       // xtal handling lift swivel in      
         "CM_ITL_IO"(ADR := 68,
             KYD_ON := "KYD".XT_HDL_SW_IN AND "PDI".MP_ENB_K9,
             KYD_OFF := NOT "KYD".XT_HDL_SW_IN OR NOT "PDI".MP_ENB_K9,
             AUTO := "DV".XT_HDL_SEQ_MOD,
             DC_ON:= "DC".XT_HDL_SW_IN AND "PDI".MP_ENB_K9,
             CON1 := "PDI".EMO AND "PDI".EMS,
             CON2 := NOT "FLT".XT_HDL_SW_ERR,
             CON3 := "PDI".LS_XT_HDL_SW_UNLOCK AND NOT "PDI".LS_XT_HDL_SW_LOCK,
             CON4 := #REL_XT_HDL_SW_IN_OK OR "DV".MP_SERVICE,   
             CON5 := NOT "DV".LS_XT_HDL_SW_IN_POS OR "DV".MP_SERVICE,  
             CON6 := ("DIS".ACT_POS_XT_HDL_LFT>=1200.0)OR "DV".MP_SERVICE,
             CON7 := "SysLog1",                     
             CON8 := "SysLog1",   
             ITL_OUT:= "STA_ITL_CAUSE",
             LT_OUT := "LT".XT_HDL_SW_IN);  

         "LT".LS_XT_HDL_SW_IN  :=  "DV".LS_XT_HDL_SW_IN_XT_POS;
         "LT".XT_HDL_SW_IN_REL :=        "PDI".EMO AND "PDI".EMS
                              AND NOT "FLT".XT_HDL_SW_ERR
                              AND "PDI".LS_XT_HDL_SW_UNLOCK AND NOT "PDI".LS_XT_HDL_SW_LOCK
                              AND (#REL_XT_HDL_SW_IN_OK OR "DV".MP_SERVICE)   
                              AND (NOT "DV".LS_XT_HDL_SW_IN_CRU_POS OR "DV".MP_SERVICE)
                              AND (("DIS".ACT_POS_XT_HDL_LFT>=1200.0)OR "DV".MP_SERVICE);

         #REL_XT_HDL_SW_IN_OK :=  (("DIS".ACT_POS_XT_HDL_LFT>1160.0) AND ("DIS".ACT_POS_XT_HDL_SW<"CNF".XT_HDL_SW_IN_TRP_POS )) 
                               OR ("PDI".LS_XT_CLP_CON AND "PDI".LS_GCH_DOOR_OP AND NOT "PDI".LS_XT_SLID_BW) 
                               OR ("PDI".LS_HOI_TOOL_INST AND "AV".TEC_FLG_ENC_POS > 100.0)
                               OR "DV".MP_SERVICE;   

         IF "LT".XT_HDL_SW_IN THEN 
           #set_speed  := "CNF_XT_HDL_SW_LZ950".SEL_SPEED;  // swivel in 
         END_IF;
         IF "LT".XT_HDL_SW_OUT THEN 
           #set_speed  := -"CNF_XT_HDL_SW_LZ950".SEL_SPEED;  // swivel out 
         END_IF;       
         IF NOT "LT".XT_HDL_SW_IN AND NOT "LT".XT_HDL_SW_OUT THEN 
           #set_speed  := 0.0; 
         END_IF;

        // Release reference set
         "LT".XT_HDL_SW_REF_RUN  := "DV".XT_HDL_SW_SET_REF_POS; ///XT_HDL_SW.READY AND NOT XT_HDL_SW.Ref_Done; //DV.XT_HDL_SW_SET_REF_POS;
         "LT".XT_HDL_SW_REF_DONE := #XT_HDL_SW.Ref_Done OR "SY".SIM_ON;                     


         #XT_HDL_SW (Enable         := ("LT".XT_HDL_SW_IN OR "LT".XT_HDL_SW_OUT OR "LT".XT_HDL_SW_REF_RUN), 
                   Pro_start     := ("LT".XT_HDL_SW_OUT OR "LT".XT_HDL_SW_IN),   
                   Speed_ext_ovr := TRUE,   
                   Ref_Start     := "LT".XT_HDL_SW_REF_RUN,
                   Ref_reset     := FALSE,
                   Reset_error   := "KYD".XT_HDL_SW_TRIP_RES,
                   Stop          := NOT "LT".XT_HDL_SW_OUT AND NOT "LT".XT_HDL_SW_IN,
                   Profil        := "CNF_XT_HDL_SW_LZ950".Profil,
                   PM_ADR_E      := INT_TO_WORD("CNF_XT_HDL_SW_LZ950".PE_ADR),                                   
                   PM_ADR_A      := INT_TO_WORD("CNF_XT_HDL_SW_LZ950".PA_ADR),                
                   Units_per_rev := "CNF_XT_HDL_SW_LZ950".UNITS_PER_REV,                       
                   Gear_ratio    := "CNF_XT_HDL_SW_LZ950".FEED_CONST,
                   Set_vel       := #set_speed); 


        //actual motor values
        //---------------------
         "AV".XT_HDL_SW_ACT_POS   := #XT_HDL_SW.Act_pos;
         "DIS".ACT_POS_XT_HDL_SW  := "AV".XT_HDL_SW_ENC_POS;   

        //actual fault
        //---------------------
         "DIS".XT_HDL_SW_ERR_CODE := #XT_HDL_SW.Error_code;        // Fehlernummer Umrichter
         "FLT".XT_HDL_SW_ERR      := #XT_HDL_SW.Error;             // Fehlerbit Umrichter
         "FLT".XT_HDL_SW_POS_REF  := NOT "LT".XT_HDL_SW_REF_DONE;   // Antrieb nicht referenziert
         "FLT".XT_HDL_SW_SLS      := #XT_HDL_SW.LS_neg OR #XT_HDL_SW.LS_pos;  // Fehler Sicherheitsendschalter



        // xtal handling lift swivel lock    
         "PDO".XT_HDL_SW_LOCK   :=  "DV".LS_XT_HDL_SW_IN_XT_POS AND NOT "LT".XT_HDL_SW_IN AND NOT "LT".XT_HDL_SW_IN AND 
                              "PDI".LS_XT_HDL_SW_UNLOCK AND NOT "KYD".XT_HDL_SW_OUT;

        // xtal handling lift swivel unlock     
         "PDO".XT_HDL_SW_UNLOCK :=  (NOT "DV".LS_XT_HDL_SW_IN_XT_POS OR "KYD".XT_HDL_SW_OUT) AND NOT "PDI".LS_XT_HDL_SW_UNLOCK;

         #REL_XT_HDL_SW_DRV    :=  "LT".XT_HDL_SW_UNLOCKED OR
                              "SysOndelay"( DIN := ("KYD".XT_HDL_SW_OUT AND "PDI".MP_ENB_K9),
                                          SetTime := 3,                         // setp. time
                                          ActTime := #sw_lock_dly,               // act. time
                                          Tick    := "SysTick1s");                // timebase (1s)

        // light signal crystal handling swivel unlock/locked     
         "LT".XT_HDL_SW_UNLOCKED := "PDI".LS_XT_HDL_SW_UNLOCK;
         "LT".XT_HDL_SW_LOCKED   := "PDI".LS_XT_HDL_SW_LOCK;

        //----------------------------------------------------------------------
        // xtal handling slidering drive   
        //----------------------------------------------------------------------
        // xtal handling sliding drive forwards
         "CM_ITL_IO"(ADR := 71,
            KYD_ON := "KYD".XT_HDL_SLID_FW AND "PDI".MP_ENB_K9,
            KYD_OFF := NOT "KYD".XT_HDL_SLID_FW OR NOT "PDI".MP_ENB_K9,
            AUTO := "DV".XT_HDL_SEQ_MOD,
            DC_ON:= "DC".XT_HDL_SLID_FW AND "PDI".MP_ENB_K9,
            CON1 := "PDI".EMO AND "PDI".EMS,
            CON2 := "PDI".LS_XT_SLID_FW,
            CON3 := NOT "PDO".XT_HDL_SLID_BW, 
            CON4 := (("PDI".LS_UP_XT_CLP_OP OR "PDI".LS_UP_XT_CLP_PLATE) AND ("PDI".LS_LO_XT_CLP_OP OR "PDI".LS_LO_XT_CLP_PLATE) AND "DV".LS_XT_HDL_SW_IN_XT_POS AND ("DIS".ACT_POS_XT_HDL_LFT>839.0)) OR 
                     ("DV".LS_XT_HDL_SW_IN_TRP_POS AND ("DV".LS_XT_HDL_LFT_DN_POS OR ("DIS".ACT_POS_XT_HDL_LFT>1120.0))) OR "DV".LS_XT_HDL_SW_OUT_MAX_POS OR 
                      //OR
                     (NOT "PDI".LS_XT_CLP_CON AND ("DIS".ACT_POS_XT_HDL_LFT>1120.0)) OR "DV".MP_SERVICE,   
            CON5 := "SysLog1",   
            CON6 := "SysLog1",                     
            CON7 := "SysLog1",    
            CON8 := "SysLog1",   
            ITL_OUT:= "STA_ITL_CAUSE",
            LT_OUT := "LT".XT_SLID_FW);

       // controller crystal handling slider forwards  
        "PDO".XT_HDL_SLID_FW  :=  "LT".XT_SLID_FW;             
        "LT".XT_SLID_FW_REL   :=      "PDI".EMO AND "PDI".EMS 
                              AND "PDI".LS_XT_SLID_FW 
                              AND NOT "PDO".XT_HDL_SLID_BW
                              AND ((("PDI".LS_UP_XT_CLP_OP OR "PDI".LS_UP_XT_CLP_PLATE) AND ("PDI".LS_LO_XT_CLP_OP OR "PDI".LS_LO_XT_CLP_PLATE) AND "DV".LS_XT_HDL_SW_IN_XT_POS AND ("DIS".ACT_POS_XT_HDL_LFT>839.0))
                                     OR ("DV".LS_XT_HDL_SW_IN_TRP_POS AND ("DV".LS_XT_HDL_LFT_DN_POS OR ("DIS".ACT_POS_XT_HDL_LFT>1120.0)))  OR "DV".LS_XT_HDL_SW_OUT_MAX_POS OR 
                                     // OR
                                     (NOT "PDI".LS_XT_CLP_CON AND ("DIS".ACT_POS_XT_HDL_LFT>1120.0)) OR "DV".MP_SERVICE);                           

       // xtal handling sliding drive backwards 
        "CM_ITL_IO"(ADR := 72,
             KYD_ON := "KYD".XT_HDL_SLID_BW AND "PDI".MP_ENB_K9,
            KYD_OFF := NOT "KYD".XT_HDL_SLID_BW OR NOT "PDI".MP_ENB_K9,
            AUTO := "DV".XT_HDL_SEQ_MOD,
            DC_ON:= "DC".XT_HDL_SLID_BW AND "PDI".MP_ENB_K9,
            CON1 := "PDI".EMO AND "PDI".EMS,
            CON2 := "PDI".LS_XT_SLID_BW,
            CON3 := NOT "PDO".XT_HDL_SLID_FW, 
            CON4 := #REL_XT_CLP_POS_OK,   
            CON5 := "SysLog1",   
            CON6 := "SysLog1",                     
            CON7 := "SysLog1",    
            CON8 := "SysLog1",   
            ITL_OUT:= "STA_ITL_CAUSE",
            LT_OUT := "LT".XT_SLID_BW);

       // controller crystal handling slider backwards  
        "PDO".XT_HDL_SLID_BW  := "LT".XT_SLID_BW; 
        "LT".XT_SLID_BW_REL   :=     "PDI".EMO AND "PDI".EMS 
                            AND "PDI".LS_XT_SLID_BW 
                            AND NOT "PDO".XT_HDL_SLID_FW
                            AND #REL_XT_CLP_POS_OK;  

        #REL_XT_CLP_POS_OK :=  (NOT "PDI".LS_XT_CLP_CON  AND ("DV".LS_XT_HDL_LFT_DN_POS OR ("DIS".ACT_POS_XT_HDL_LFT>620.0)))        // without clamp
                           OR ("PDI".LS_XT_CLP_CON AND (("PDI".LS_UP_XT_CLP_CL AND "PDI".LS_LO_XT_CLP_CL) OR ("PDI".LS_UP_XT_CLP_SAVE AND "PDI".LS_LO_XT_CLP_SAVE) OR "DV".LS_XT_HDL_SW_IN_TRP_POS) 
                           AND "PDI".LS_XT_SLID_BW AND "PDI".LS_XT_TILT_90 AND ("DIS".ACT_POS_XT_HDL_LFT>620.0))   // takeover cystal 
                           OR (NOT "PDI".LS_XT_TILT_75 AND "DV".LS_XT_ACP_LFT_UPR_POS) // lift up to 1550mm position ready to swivel out to 56?
                           OR "DV".LS_XT_HDL_SW_OUT_MAX_POS
                           OR "DV".MP_SERVICE;          

       //light signal for positions  
        "LT".LS_XT_SLID_FW       :=   NOT "PDI".LS_XT_SLID_FW AND NOT "PDI".LS_XT_SLID_MID  AND "PDI".LS_XT_SLID_BW;          
        "LT".LS_XT_SLID_MID      :=   "PDI".LS_XT_SLID_MID AND "PDI".LS_XT_SLID_FW AND "PDI".LS_XT_SLID_BW;           
        "LT".LS_XT_SLID_BW       :=   NOT "PDI".LS_XT_SLID_BW AND "PDI".LS_XT_SLID_FW AND NOT "PDI".LS_XT_SLID_MID;         


       //----------------------------------------------------------------------
       // xtal handling tilt drive       
       //---------------------------------------------------------------------- 
       // xtal handling tilt drive forwards (to 75?
        "CM_ITL_IO"(ADR := 73,
            KYD_ON := "KYD".XT_CLP_TILT_75 AND "PDI".MP_ENB_K9,
            KYD_OFF := NOT "KYD".XT_CLP_TILT_75 OR NOT "PDI".MP_ENB_K9,
            AUTO := "DV".XT_HDL_SEQ_MOD,
            DC_ON:= "DC".XT_CLP_TILT_75 AND "PDI".MP_ENB_K9,
            CON1 := "PDI".EMO AND "PDI".EMS,
            CON2 := NOT "PDI".LS_XT_TILT_75,
            CON3 := NOT "PDO".XT_CLP_TILT_BW, 
            CON4 := #REL_XT_CLP_TILT_POS_OK OR "DV".MP_SERVICE,                
            CON5 := "SysLog1",   
            CON6 := "SysLog1",                     
            CON7 := "SysLog1",    
            CON8 := "SysLog1",   
            ITL_OUT:= "STA_ITL_CAUSE",
            LT_OUT := "LT".XT_TILT_75);

       // controller crystal handling slider forwards  
        "PDO".XT_CLP_TILT_FW  := "LT".XT_TILT_75;
        "LT".XT_TILT_75_REL   :=         "PDI".EMO AND "PDI".EMS 
                             AND NOT "PDI".LS_XT_TILT_75 
                             AND NOT "PDO".XT_CLP_TILT_BW 
                             AND (#REL_XT_CLP_TILT_POS_OK OR "DV".MP_SERVICE);

        #REL_XT_CLP_TILT_POS_OK :=  "DV".LS_XT_HDL_SW_IN_XT_POS AND "PDI".LS_XT_SLID_MID;


       // xtal handling tilt drive backwards (to 90?  
        "CM_ITL_IO"(ADR := 74,
            KYD_ON := "KYD".XT_CLP_TILT_90 AND "PDI".MP_ENB_K9,
            KYD_OFF := NOT "KYD".XT_CLP_TILT_90 OR NOT "PDI".MP_ENB_K9,
            AUTO := "DV".XT_HDL_SEQ_MOD,
            DC_ON:= "DC".XT_CLP_TILT_90 AND "PDI".MP_ENB_K9,
            CON1 := "PDI".EMO AND "PDI".EMS,
            CON2 := NOT "PDI".LS_XT_TILT_90,
            CON3 := NOT "PDO".XT_CLP_TILT_FW, 
            CON4 := "DV".LS_XT_HDL_SW_IN_TRP_POS OR "DV".MP_SERVICE,         
            CON5 := "SysLog1",   
            CON6 := "SysLog1",                     
            CON7 := "SysLog1",    
            CON8 := "SysLog1",   
            ITL_OUT:= "STA_ITL_CAUSE",
            LT_OUT := "LT".XT_TILT_90);

       // controller crystal handling slider backwards  
        "PDO".XT_CLP_TILT_BW  :=  "LT".XT_TILT_90;
        "LT".XT_TILT_90_REL   :=      "PDI".EMO AND "PDI".EMS 
                             AND NOT "PDI".LS_XT_TILT_90 
                             AND NOT "PDO".XT_CLP_TILT_BW 
                             AND ("DV".LS_XT_HDL_SW_IN_TRP_POS OR "DV".MP_SERVICE);

       // Open Brake    
        "PDO".XT_CLP_TILT_BRK:= "PDO".XT_CLP_TILT_FW OR "PDO".XT_CLP_TILT_BW;  

       //light signal for positions  
        "LT".LS_XT_TILT_90  :=   "PDI".LS_XT_TILT_90 AND NOT "PDI".LS_XT_TILT_75;
        "LT".LS_XT_TILT_75  :=   "PDI".LS_XT_TILT_75 AND NOT "PDI".LS_XT_TILT_90;

       //----------------------------------------------------------------------
       // xtal handling xtal clamps      
       //---------------------------------------------------------------------- 
       // xtal handling clamps above open
        "CM_ITL_IO"(ADR := 75,
            KYD_ON := "KYD".XT_CLP_ABV_OP AND "PDI".MP_ENB_K9,
            KYD_OFF := NOT "KYD".XT_CLP_ABV_OP OR NOT "PDI".MP_ENB_K9,
            AUTO := "DV".XT_HDL_SEQ_MOD,
            DC_ON:= "DC".XT_CLP_ABV_OP AND "PDI".MP_ENB_K9,
            CON1 := "PDI".EMO AND "PDI".EMS,
            CON2 := "PDI".LS_XT_CLP_CON,         
            CON3 := NOT "PDO".XT_CLP_ABV_CL,
            CON4 := NOT "PDI".LS_UP_XT_CLP_OP, 
            CON5 := "PDI".LS_XT_TILT_90 OR "DV".MP_SERVICE,   
            CON6 := NOT "PDI".LS_UP_XT_CLP_PLATE,                     
            CON7 := "SysLog1",    
            CON8 := "SysLog1",   
            ITL_OUT:= "STA_ITL_CAUSE",
            LT_OUT := "PDO".XT_CLP_ABV_OP);

       // xtal handling clamps above close   
        "CM_ITL_IO"(ADR := 76,
            KYD_ON := "KYD".XT_CLP_ABV_CL AND "PDI".MP_ENB_K9,
            KYD_OFF := NOT "KYD".XT_CLP_ABV_CL OR NOT "PDI".MP_ENB_K9 ,
            AUTO := "DV".XT_HDL_SEQ_MOD,
            DC_ON:= "DC".XT_CLP_ABV_CL AND "PDI".MP_ENB_K9,
            CON1 := "PDI".EMO AND "PDI".EMS,
            CON2 := "PDI".LS_XT_CLP_CON,         
            CON3 := NOT "PDO".XT_CLP_ABV_OP,
            CON4 := NOT "PDI".LS_UP_XT_CLP_CL, 
            CON5 := NOT "PDI".LS_UP_XT_CLP_PLATE,   
            CON6 := "SysLog1",                     
            CON7 := "SysLog1",    
            CON8 := "SysLog1",   
            ITL_OUT:= "STA_ITL_CAUSE",
            LT_OUT := "PDO".XT_CLP_ABV_CL);

        "LT".UP_XT_CLP_CL := "PDO".XT_CLP_ABV_CL; 
        "LT".UP_XT_CLP_OP := "PDO".XT_CLP_ABV_OP; 
        "LT".UP_XT_CLP_CL_REL:= "PDI".EMO AND "PDI".EMS AND "PDI".LS_XT_CLP_CON AND NOT "PDO".XT_CLP_ABV_OP AND NOT "PDI".LS_UP_XT_CLP_CL AND NOT "PDI".LS_UP_XT_CLP_PLATE;
        "LT".UP_XT_CLP_OP_REL:= "PDI".EMO AND "PDI".EMS AND "PDI".LS_XT_CLP_CON AND NOT "PDO".XT_CLP_ABV_CL AND NOT "PDI".LS_UP_XT_CLP_OP AND ("PDI".LS_XT_TILT_90 OR "DV".MP_SERVICE) 
                              AND NOT "PDI".LS_UP_XT_CLP_PLATE; 

       // xtal handling clamps below open 
        "CM_ITL_IO"(ADR := 77,
            KYD_ON := ("KYD".XT_CLP_BLW_OP  OR ("KYD".XT_CLP_ABV_OP AND NOT "PDI".LS_LO_XT_CLP_PLATE)) AND "PDI".MP_ENB_K9,
            KYD_OFF := (NOT "KYD".XT_CLP_BLW_OP AND NOT "KYD".XT_CLP_ABV_OP) OR NOT "PDI".MP_ENB_K9 ,
            AUTO := "DV".XT_HDL_SEQ_MOD,
            DC_ON:= "DC".XT_CLP_BLW_OP AND "PDI".MP_ENB_K9,
            CON1 := "PDI".EMO AND "PDI".EMS,
            CON2 := "PDI".LS_XT_CLP_CON,                  
            CON3 := NOT "PDO".XT_CLP_BLW_CL,
            CON4 := NOT "PDI".LS_LO_XT_CLP_OP, 
            CON5 := "PDI".LS_XT_TILT_90 OR "DV".MP_SERVICE,   
            CON6 := NOT "PDI".LS_LO_XT_CLP_PLATE,                     
            CON7 := "SysLog1",    
            CON8 := "SysLog1",   
            ITL_OUT:= "STA_ITL_CAUSE",
            LT_OUT := "PDO".XT_CLP_BLW_OP);

       // xtal handling clamps below close   
        "CM_ITL_IO"(ADR := 78,
            KYD_ON := ("KYD".XT_CLP_BLW_CL OR ("KYD".XT_CLP_ABV_CL AND NOT "PDI".LS_LO_XT_CLP_PLATE)) AND "PDI".MP_ENB_K9,
            KYD_OFF := (NOT "KYD".XT_CLP_BLW_CL AND NOT "KYD".XT_CLP_ABV_CL)OR NOT "PDI".MP_ENB_K9 ,
            AUTO := "DV".XT_HDL_SEQ_MOD,
            DC_ON:= "DC".XT_CLP_BLW_CL AND "PDI".MP_ENB_K9,
            CON1 := "PDI".EMO AND "PDI".EMS,
            CON2 := "PDI".LS_XT_CLP_CON,         
            CON3 := NOT "PDO".XT_CLP_BLW_OP,
            CON4 := NOT "PDI".LS_LO_XT_CLP_CL, 
            CON5 := NOT "PDI".LS_LO_XT_CLP_PLATE,   
            CON6 := "SysLog1",                     
            CON7 := "SysLog1",    
            CON8 := "SysLog1",                  
            ITL_OUT:= "STA_ITL_CAUSE",
            LT_OUT := "PDO".XT_CLP_BLW_CL);  

        "LT".LO_XT_CLP_CL := "PDO".XT_CLP_BLW_CL; 
        "LT".LO_XT_CLP_OP := "PDO".XT_CLP_BLW_OP; 
        "LT".LO_XT_CLP_CL_REL := "PDI".EMO AND "PDI".EMS AND NOT "PDO".XT_CLP_BLW_OP AND NOT "PDI".LS_LO_XT_CLP_CL AND NOT "PDI".LS_LO_XT_CLP_PLATE;
        "LT".LO_XT_CLP_OP_REL := "PDI".EMO AND "PDI".EMS AND "PDI".LS_XT_CLP_CON AND NOT "PDO".XT_CLP_BLW_CL AND NOT "PDI".LS_LO_XT_CLP_OP AND ("PDI".LS_XT_TILT_90 OR "DV".MP_SERVICE) 
                              AND NOT "PDI".LS_LO_XT_CLP_PLATE;  

       //light signal for positions    
        "LT".LS_UP_XT_CLP_CL           :=   "PDI".LS_UP_XT_CLP_CL AND NOT "PDI".LS_UP_XT_CLP_OP;           
        "LT".LS_UP_XT_CLP_OP           :=   "PDI".LS_UP_XT_CLP_OP AND NOT "PDI".LS_UP_XT_CLP_CL;    
        "LT".LS_LO_XT_CLP_CL           :=   "PDI".LS_LO_XT_CLP_CL AND NOT "PDI".LS_LO_XT_CLP_OP;  
        "LT".LS_LO_XT_CLP_OP           :=   "PDI".LS_LO_XT_CLP_OP AND NOT "PDI".LS_LO_XT_CLP_CL;  
       //LT.UP_XT_CLP_SAVE         :=   PDI.LS_UP_XT_CLP_SAVE;
       //LT.LO_XT_CLP_SAVE         :=   PDI.LS_LO_XT_CLP_SAVE;

       //OPEN crystal clamp above/below brake
        "PDO".XT_CLP_ABV_BRK := "PDO".XT_CLP_ABV_CL OR "PDO".XT_CLP_ABV_OP;    
        "PDO".XT_CLP_BLW_BRK := "PDO".XT_CLP_BLW_CL OR "PDO".XT_CLP_BLW_OP;

       // reset controller crystal clamp above/below
        "PDO".XT_CLP_ABV_RST := "KYD".XT_CLP_ABV_RST;
        "PDO".XT_CLP_BLW_RST := "KYD".XT_CLP_BLW_RST;


       //----------------------------------------------------------------------
       // xtal drop out protection
       //---------------------------------------------------------------------- 
       #rel_man_move := ("APC".STATUS = "APC".IDLE) AND "DV".APS_GCH_DELAYED;
       //open/close crystal drop out protection of gate chamber manually
       //---------------------------------------------------------------
       IF "PDI".LS_GCH_DOOR_OP OR #rel_man_move THEN     //open/close drop out protection manually only when door is open
         "LT".XT_DRP_OUT_PRT_ENB   :=  TRUE;          //set enable light flag
         //open drop out protection
         //------------------------
         IF "KYD".OP_XT_DRP_OUT_PRT  OR "DC".OP_XT_DRP_OUT_PRT THEN
             "PDO".XT_DRP_OUT_PRT_OP   :=  TRUE;
             "PDO".XT_DRP_OUT_PRT_CL   :=  FALSE;
         //close drop out protection
         //-------------------------
         ELSIF "KYD".CL_XT_DRP_OUT_PRT OR "DC".CL_XT_DRP_OUT_PRT THEN
             "PDO".XT_DRP_OUT_PRT_OP   :=  FALSE;
             "PDO".XT_DRP_OUT_PRT_CL   :=  TRUE;        
         END_IF;
       ELSE
         "LT".XT_DRP_OUT_PRT_ENB   :=  FALSE;      //reset enable light flag
       END_IF;

      //open/close crystal drop out protection of gate chamber automatically
      //--------------------------------------------------------------------
       IF "SysTick1s" THEN 
         IF "PDI".LS_GCH_DOOR_CL AND NOT #rel_man_move  THEN            //gate chamber door closed
             IF "DV".APS_GCH_DELAYED THEN             //atmospheric pressure
                 //close drop out protection 
                 //-------------------------
                 IF ("DV".APS_GCH_DELAYED <> #gch_prs_prev) THEN    //compare pressure status from previous cycle
                     "PDO".XT_DRP_OUT_PRT_CL   :=  TRUE;
                     "PDO".XT_DRP_OUT_PRT_OP   :=  FALSE;
                 END_IF;
             ELSE                            //vacuum pressure
                 //open drop out protection 
                 //------------------------
                 "PDO".XT_DRP_OUT_PRT_CL   :=  FALSE;
                 "PDO".XT_DRP_OUT_PRT_OP   :=  TRUE;
             END_IF;
         END_IF;       

         #gch_prs_prev    :=  "DV".APS_GCH_DELAYED;  //store pressure status of gate chamber in 1 sec intervall

       END_IF;

      //set light flag drop out protection opened
      //-----------------------------------------
       "LT".XT_DRP_OUT_PRT_OP    :=  "PDI".XT_DRP_OUT_PRT_1_OP AND 
                                 "PDI".XT_DRP_OUT_PRT_2_OP AND
                                 "PDI".XT_DRP_OUT_PRT_3_OP AND
                                 "PDI".XT_DRP_OUT_PRT_4_OP;

      //set light flag drop out protection closed
      //-----------------------------------------
       "LT".XT_DRP_OUT_PRT_CL    :=  "PDI".XT_DRP_OUT_PRT_1_CL AND 
                                 "PDI".XT_DRP_OUT_PRT_2_CL AND
                                 "PDI".XT_DRP_OUT_PRT_3_CL AND
                                 "PDI".XT_DRP_OUT_PRT_4_CL;
      //evaluate status of drop out protection
      //--------------------------------------
       "FLT".XT_DRP_OUT_PRT_OP   :=  "SysOndelay" (DIN     :=  ("PDO".XT_DRP_OUT_PRT_OP XOR "LT".XT_DRP_OUT_PRT_OP) AND NOT "LT".MAG_ON,
                                             SetTime :=  60,      
                                             Tick    :=  "SysTick100ms",                 
                                             ActTime :=  #op_flt_dly);

       "FLT".XT_DRP_OUT_PRT_CL   :=  "SysOndelay" (DIN     :=  ("PDO".XT_DRP_OUT_PRT_CL XOR "LT".XT_DRP_OUT_PRT_CL) AND NOT "LT".MAG_ON,
                                             SetTime :=  60,      
                                             Tick    :=  "SysTick100ms",                 
                                             ActTime :=  #cl_flt_dly);

      //crystal clamp have plate

       "LT".LS_UP_XT_CLP_PLATE := "PDI".LS_UP_XT_CLP_PLATE;



      //Write postion values for mobile panel
      //--------------------------------------------

       IF "DIS".ACT_POS_XT_HDL_LFT<11.0 THEN
           "STA".XT_HDL_LFT_POS  := 0;
          ELSIF "DIS".ACT_POS_XT_HDL_LFT>2900.0 THEN 
           "STA".XT_HDL_LFT_POS  := 100;
       ELSE    
           "STA".XT_HDL_LFT_POS  :=  REAL_TO_INT("DIS".ACT_POS_XT_HDL_LFT/30.0);   
       END_IF;

       IF NOT "PDI".LS_XT_SLID_BW THEN 
           "STA".XT_HDL_SLID_POS := 0;
          ELSIF "PDI".LS_XT_SLID_MID THEN
           "STA".XT_HDL_SLID_POS := 50;
          ELSIF NOT "PDI".LS_XT_SLID_FW THEN   
           "STA".XT_HDL_SLID_POS := 100;
       END_IF;
END_FUNCTION_BLOCK

FUNCTION_BLOCK "BM_XT_HDL_SEQ"   // FB61, SCL
{ S7_Optimized_Access := 'FALSE' }
VERSION : 0.0
// --------------------------------------------------------------------------------
//     program     :   BM_XT_HDL_SEQ
//     description :   Sequencer crystal handling
//     name        :   John Wang
//     date        :   23.11.2018
//   
//     revision    :
//     name        :
//     date        :    
//                     (c)PVA CGS GmbH
//     --------------------------------------------------------------------------------
   VAR
      Dummy : Bool;
      end_of_step : Bool;
      arb_seq : Bool;
      "step" : Int;
      next_step : Int;
      i : Int;
      j : Int;
      STEP_MSG : Int;
   END_VAR
BEGIN


        "LT".XT_HDL_SEQ_MOD := "LT".XT_HDL_SEQ_XT_OUT OR "LT".XT_HDL_SEQ_LD_CRU OR "LT".XT_HDL_SEQ_HDL_HZ; // Auto mode of crystal handling
        "STA".OP_MSG_HDL_SEQ  := #STEP_MSG;  

      //set step to abort docking sequence
      //----------------------------------
      IF (#arb_seq AND (#step <> 1000)) THEN
         #step    := 1000;
      END_IF;

           //sequence steps
      //--------------
      CASE #step OF 

      //-----------------------------------------------------------                 
      // initialisation step and select sub sequence
      //-----------------------------------------------------------
      0:                                                           
               IF #next_step = #step THEN
                  "LT".XT_HDL_SEQ_XT_OUT  := FALSE;                           
                  "LT".XT_HDL_SEQ_LD_CRU  := FALSE;                           
                  "LT".XT_HDL_SEQ_HDL_HZ  := FALSE;                           
                  #next_step := 10;                                                  
               END_IF;


               IF "KYD".XT_HDL_SEQ_XT_OUT AND "PDI".MP_ENB_K9 THEN                    
                   #end_of_step := true; 
                   #next_step := 10;
                   "LT".XT_HDL_SEQ_XT_OUT  := TRUE;
                   "KYD".XT_HDL_SEQ_XT_OUT := FALSE;                           
               END_IF;

               IF "KYD".XT_HDL_SEQ_LD_CRU AND "PDI".MP_ENB_K9 THEN                    
                   #end_of_step := true; 
                   #next_step := 300;
                   "LT".XT_HDL_SEQ_LD_CRU  := TRUE; 
                   "KYD".XT_HDL_SEQ_LD_CRU := FALSE;                           
               END_IF;

               IF "KYD".XT_HDL_SEQ_HDL_HZ AND "PDI".MP_ENB_K9 THEN                    
                   #end_of_step := true;
                   #next_step := 600; 
                   "LT".XT_HDL_SEQ_HDL_HZ := TRUE; 
                   "KYD".XT_HDL_SEQ_HDL_HZ := FALSE;                           
               END_IF;


      //-----------------------------------------------------------                 
      // 1.Step : Check start conditions
      //-----------------------------------------------------------
      10:                                                           
               IF #next_step = #step THEN
                   #STEP_MSG := 10;
                   "APC".TI[6] := 0; 

               END_IF;

               "DC".XT_HDL_LFT_UP  := "DIS".ACT_POS_XT_HDL_LFT <500.0;    // 300mm;      // Lift in upper safe position
               "DC".XT_HDL_SW_OUT  := "DIS".ACT_POS_XT_HDL_SW >10.0;        // swivel drive in outer position
               "DC".XT_HDL_SLID_BW := NOT "PDI".LS_XT_SLID_BW;                   // slider drive in back position


               IF NOT "DC".XT_HDL_LFT_UP AND NOT "DC".XT_HDL_SW_OUT AND NOT "DC".XT_HDL_SLID_BW AND "PDI".LS_GCH_DOOR_OP THEN
                  "LT".XT_HDL_OP_CONT := True;                       // Question: Is crystall carriage in postion?                   
                  IF "KYD".XT_HDL_OP_CONT THEN                       // IF Operator confirm carriage pos. continue                    
                     #end_of_step := true; 
                     "KYD".XT_HDL_OP_CONT := FALSE;    
                     "LT".XT_HDL_OP_CONT  := FALSE;                         
                  END_IF;
               END_IF;                                    

               #next_step := 20; 

      //-----------------------------------------------------------                 
      // 2.step XT-Handling lift drive in takeover position 350 mm
      //-----------------------------------------------------------
      20:                                                           
               IF #next_step = #step THEN
                   #STEP_MSG  := 20;
                   "APC".TI[6] := 0;                                                  
               END_IF;


              IF ABS("DIS".ACT_POS_XT_HDL_LFT-350.0)>1.0 THEN
                  "DC".XT_HDL_LFT_DN   := TRUE;
                  ELSE
                  "DC".XT_HDL_LFT_DN  := FALSE;
              END_IF;

         //    DC.XT_HDL_LFT_DN  := ABS(DIS.ACT_POS_XT_HDL_LFT-10.0)<1.0;         // Lift in takeover position
               "DC".XT_HDL_LFT_FAST := "DC".XT_HDL_LFT_DN AND "DIS".ACT_POS_XT_HDL_LFT <2495.0;

              IF "APC".TI[6]> 3 AND NOT "DC".XT_HDL_LFT_DN THEN                    
                   #end_of_step := true;                            
              END_IF;                                    

               #next_step := 30; 


      //-------------------------------------------------------------                
      //  3.step XT-Handling swivel-in drive in takeover position 56?
      //-------------------------------------------------------------
      30:                                                           
              IF #next_step = #step THEN
                   #STEP_MSG  := 30;
                   "APC".TI[6] := 0;                                                  
              END_IF;


              IF ABS("DIS".ACT_POS_XT_HDL_SW-56.0)>0.1 THEN
                 "DC".XT_HDL_SW_IN   := TRUE;
                 ELSE
                 "DC".XT_HDL_SW_IN  := FALSE;
              END_IF;

              IF "APC".TI[6]> 3 AND NOT "DC".XT_HDL_SW_IN THEN                    
                  #end_of_step := true;                            
              END_IF;                                    
                  #next_step := 40;


      //-----------------------------------------------------------                 
      // 4.step XT-HDL Sliding drive forward in takeover position
      //-----------------------------------------------------------
      40:                                                           
               IF #next_step = #step THEN
                   #STEP_MSG  := 40;
                   "APC".TI[6] := 0;                                                  
               END_IF;
                "DC".XT_HDL_SLID_FW := NOT "PDI".LS_XT_SLID_FW;            // slider drive in work position 

               IF "APC".TI[6]> 3 AND NOT "DC".XT_HDL_SLID_FW THEN                    
                  #end_of_step := true;                            
               END_IF;                                    
                  #next_step := 50;

      //-----------------------------------------------------------                 
      // 5.step XT-Handling lift drive in crystal position 1500 mm 
      //-----------------------------------------------------------
      50:                                                           
               IF #next_step = #step THEN
                   #STEP_MSG  := 50;
                   "APC".TI[6] := 0;                                                  
               END_IF;

               IF ABS("DIS".ACT_POS_XT_HDL_LFT - 1500.0) > 1.0 THEN
                  "DC".XT_HDL_LFT_UP   := TRUE;                             // Lift in crystal middle position
                  ELSE
                  "DC".XT_HDL_LFT_UP  := FALSE;
               END_IF;

               // setze langsame Speed ein f黵 einstecken des St鋟blisteckers

               "DC".XT_HDL_LFT_FAST := "DC".XT_HDL_LFT_UP AND "DIS".ACT_POS_XT_HDL_LFT >355.0;

               IF "APC".TI[6]> 3 AND NOT "DC".XT_HDL_LFT_UP THEN                    
                  #end_of_step := true;                            
               END_IF;                                    
                  #next_step := 60; 

      //-----------------------------------------------------------                 
      // 6.step XT-HDL Sliding drive backward in home position     
      //-----------------------------------------------------------
      60:                                                           
               IF #next_step = #step THEN
                   #STEP_MSG  := 60;
                   "APC".TI[6] := 0;                                                  
               END_IF;

               IF "PDI".LS_XT_CLP_CON THEN 
                 "DC".XT_HDL_SLID_BW := NOT "PDI".LS_XT_SLID_BW; 
               END_IF;  

               IF "APC".TI[6]> 3 AND NOT "DC".XT_HDL_SLID_BW THEN                    
                  #end_of_step := true;                            
               END_IF;                                        
                  #next_step := 70; 


      //-----------------------------------------------------------                 
      // 7.step XT-Handling swivel-in drive to gate chamber 145?
      //-----------------------------------------------------------
     70:                                                           
               IF #next_step = #step THEN
                   #STEP_MSG  := 70;
                   "APC".TI[6] := 0;                                                  
               END_IF;

               "DC".XT_HDL_SW_IN   := "DIS".ACT_POS_XT_HDL_SW < 145.0 OR NOT "PDI".LS_XT_HDL_SW_LOCK;            
               "DC".XT_HDL_SW_LOCK := NOT "PDI".LS_XT_HDL_SW_LOCK; 

               IF "APC".TI[6]> 3 AND NOT "DC".XT_HDL_SW_IN AND "PDI".LS_XT_HDL_SW_LOCK THEN                    
                  #end_of_step := true;                            
               END_IF;                                      
                  #next_step := 80; 

      //-----------------------------------------------------------                 
      // 8.step Open drop out protection
      //-----------------------------------------------------------
      80:                                                           
              IF #next_step = #step THEN
                   #STEP_MSG  := 80;
                   "APC".TI[6] := 0;                                                  
              END_IF;

              IF "PDI".LS_XT_HDL_SW_LOCK THEN 
                 "DC".OP_XT_DRP_OUT_PRT:= NOT "LT".XT_DRP_OUT_PRT_OP;
              END_IF;

              IF "APC".TI[6]> 3 AND NOT "DC".OP_XT_DRP_OUT_PRT AND NOT "FLT".XT_DRP_OUT_PRT_OP THEN                    
                  #end_of_step := true;                            
              END_IF;                                    
                  #next_step := 90;

      //-----------------------------------------------------------------                 
      // 9.step XT-HDL Sliding drive forward in crystal takeover position
      //-----------------------------------------------------------------
      90:                                                           
               IF #next_step = #step THEN
                   #STEP_MSG  := 90;  
                   "APC".TI[6] := 0;                                                  
               END_IF;

               "DC".XT_HDL_SLID_FW := NOT "PDI".LS_XT_SLID_FW ;

               IF "APC".TI[6]> 3 AND NOT "DC".XT_HDL_SLID_FW THEN                    
                  #end_of_step := true;                            
               END_IF;                                    
                  #next_step := 100;


      //-----------------------------------------------------------                 
      // 10.step XT-Handling lift drive down to crystal takeover position (h鋘disch) 1480 2mm vor Teller 
      //-----------------------------------------------------------
      100:                                                           
              IF #next_step = #step THEN
                   #STEP_MSG  := 100;
                   "APC".TI[6] := 0;                                                  
              END_IF;

              IF "LT".XT_DRP_OUT_PRT_OP AND "PDI".LS_XT_SLID_FW THEN 
                 "LT".XT_HDL_CLP_OP_CONT := TRUE;                   //Question: Is crystal clamp in safety work position? 

                IF "KYD".XT_HDL_CLP_OP_CONT THEN                       // If Operator per mob. panel confirm  pos. continue                    
                     #end_of_step := true; 
                     "KYD".XT_HDL_CLP_OP_CONT := FALSE;    
                     "LT".XT_HDL_CLP_OP_CONT  := FALSE;                         
                END_IF;
              END_IF;                                    

              IF "APC".TI[6]> 3 AND NOT "LT".XT_HDL_CLP_OP_CONT THEN                    
                  #end_of_step := true;                            
              END_IF;                     
                  #next_step := 110;


      //-----------------------------------------------------------                 
      // 11.step crystal clamp closing                                       
      //-----------------------------------------------------------
      110:                                                           
               IF #next_step = #step THEN
                   #STEP_MSG  := 110;
                   "APC".TI[6] := 0;                                                  
               END_IF;

               "DC".XT_CLP_ABV_CL  :=  NOT "PDI".LS_UP_XT_CLP_CL OR NOT "PDI".LS_UP_XT_CLP_SAVE;    // noch zu fragen
               "DC".XT_CLP_BLW_CL  :=  NOT "PDI".LS_LO_XT_CLP_CL OR NOT "PDI".LS_LO_XT_CLP_SAVE; 

               IF "APC".TI[6]> 3 AND NOT "DC".XT_CLP_ABV_CL AND NOT "DC".XT_CLP_BLW_CL THEN                    
                  #end_of_step := true;                            
               END_IF;                                    
                  #next_step := 120;

      //-----------------------------------------------------------                 
      // 12.Require cut crystal neck manually und confirm it
      //-----------------------------------------------------------
      120:                                                           
               IF #next_step = #step THEN
                  #STEP_MSG  := 120;
                   "APC".TI[6] := 0;                                                    
               END_IF;

                 "LT".XT_HDL_CUT_OP_CONT := TRUE; 

               IF "KYD".XT_HDL_CUT_OP_CONT  THEN                    
                   #end_of_step := true;
                   "LT".XT_HDL_CUT_OP_CONT  := FALSE;  
                   "KYD".XT_HDL_CUT_OP_CONT := FALSE; 
               END_IF;                                    

               IF "APC".TI[6]> 3 AND NOT "LT".XT_HDL_CUT_OP_CONT THEN                    
                  #end_of_step := true;                            
               END_IF;        
                  #next_step := 130; 

      //-----------------------------------------------------------                 
      // 13.step XT-HDL Sliding drive backward in middle position            
      //-----------------------------------------------------------
      130:                                                           

               IF #next_step = #step THEN
                   #STEP_MSG  := 130;
                   "APC".TI[6] := 0;                                                  
               END_IF;
                  "DC".XT_HDL_SLID_BW := NOT "PDI".LS_XT_SLID_MID;   

               IF "APC".TI[6]> 3 AND NOT "DC".XT_HDL_SLID_BW THEN                    
                  #end_of_step := true;                            
               END_IF;                                        
                  #next_step := 140; 

      //-----------------------------------------------------------                 
      // 14.step XT-HDL tilt drive forwards in 75?position        
      //-----------------------------------------------------------
      140:                                                           
               IF #next_step = #step THEN
                   #STEP_MSG  := 140;
                   "APC".TI[6] := 0;                                                  
               END_IF;            

                  "DC".XT_CLP_TILT_75 := "PDI".LS_XT_TILT_75;

               IF "APC".TI[6]> 3 AND NOT "DC".XT_CLP_TILT_75 THEN                    
                  #end_of_step := true;                            
               END_IF;                                   
               #next_step := 150;

      //------------------------------------------------------------------------                 
      // 15.step XT-Handling lift drive in upper position in gate chamber 1550 mm         
      //------------------------------------------------------------------------
      150:                                                           
               IF #next_step = #step THEN
                   #STEP_MSG  := 150;
                   "APC".TI[6] := 0;                                                  
               END_IF;             

               IF ABS("DIS".ACT_POS_XT_HDL_LFT-1550.0) > 1.0 THEN 
                  "DC".XT_HDL_LFT_UP := TRUE;
                  ELSE
                  "DC".XT_HDL_LFT_UP := FALSE;
               END_IF;

               IF "APC".TI[6]> 3 AND NOT "DC".XT_HDL_LFT_UP THEN 
                   #end_of_step := true;                            
               END_IF;                                   
                   #next_step := 160;

      //-----------------------------------------------------------                 
      // 16.step XT-HDL Sliding drive backward in home position     
      //-----------------------------------------------------------
      160:                                                           
               IF #next_step = #step THEN
                   #STEP_MSG  := 160;
                   "APC".TI[6] := 0;                                                  
               END_IF;

              "DC".XT_HDL_SLID_BW := NOT "PDI".LS_XT_SLID_BW;   

               IF "APC".TI[6]> 3 AND NOT "DC".XT_HDL_SLID_BW THEN                    
                  #end_of_step := true;                             
              END_IF;                                    

               #next_step := 170;

      //-----------------------------------------------------------                 
      // 17.step XT-Handling swivel drive to takeover position   56?   
      //-----------------------------------------------------------
      170:                                                           
               IF #next_step = #step THEN
                   #STEP_MSG  := 170;
                   "APC".TI[6] := 0;                                                  
               END_IF;

              IF ABS("DIS".ACT_POS_XT_HDL_SW-56.0)>0.1 THEN
                 "DC".XT_HDL_SW_OUT   := TRUE;
                 ELSE
                 "DC".XT_HDL_SW_OUT  := FALSE;
              END_IF;

              IF "APC".TI[6]> 3 AND NOT "DC".XT_HDL_SW_OUT THEN                    
                  #end_of_step := true;                            
              END_IF;  
                  #next_step := 180;

      //-----------------------------------------------------------                 
      // 18.step XT-HDL tilt drive backwards in 90?position            
      //-----------------------------------------------------------
      180:                                                           

               IF #next_step = #step THEN
                   #STEP_MSG  := 180;
                   "APC".TI[6] := 0;                                                  
               END_IF;            
                  "DC".XT_CLP_TILT_90 := "PDI".LS_XT_TILT_90;
               IF "APC".TI[6]> 3 AND NOT "DC".XT_CLP_TILT_90 THEN                    
                  #end_of_step := true;                            
               END_IF;                                   
                  #next_step := 190;

      //-----------------------------------------------------------                 
      // 19.step XT-HDL Sliding drive fordward in takeover position     
      //-----------------------------------------------------------
      190:                                                           
               IF #next_step = #step THEN
                   #STEP_MSG  := 190;
                   "APC".TI[6] := 0;                                                  
               END_IF;
                  "DC".XT_HDL_SLID_FW := NOT "PDI".LS_XT_SLID_FW;   
               IF "APC".TI[6]> 3 AND NOT "DC".XT_HDL_SLID_FW THEN                    
                  #end_of_step := true;                            
               END_IF;                                        
                  #next_step := 200;

      //-----------------------------------------------------------                 
      // 20.step XT-Handling lift drive down to takeover position 350 mm     
      //-----------------------------------------------------------
      200:                                                           
               IF #next_step = #step THEN
                   #STEP_MSG  := 200;
                   "APC".TI[6] := 0;                                                  
               END_IF;

               IF "DIS".ACT_POS_XT_HDL_LFT > 350.0 THEN
                  "DC".XT_HDL_LFT_DN   := TRUE;                             
                  ELSE
                  "DC".XT_HDL_LFT_DN  := FALSE;
               END_IF;
             // setze langsamer Speed ein f黵 ausstecken des St鋟blisteckers

             //  DC.XT_HDL_LFT_FAST := DC.XT_HDL_LFT_DN AND DIS.ACT_POS_XT_HDL_LFT >400.0;

               IF "APC".TI[6]> 3 AND NOT "DC".XT_HDL_LFT_DN THEN 
                   #end_of_step := true;                            
               END_IF;                                        
                   #next_step := 210;

      //-----------------------------------------------------------                 
      // 21.step XT-HDL Sliding drive backwards in home position      
      //-----------------------------------------------------------
      210:                                                           

              IF #next_step = #step THEN
                   #STEP_MSG  := 210;
                   "APC".TI[6] := 0;                                                  
              END_IF;

              IF NOT "PDI".LS_XT_CLP_CON THEN 
                 "DC".XT_HDL_SLID_BW := NOT "PDI".LS_XT_SLID_BW; 
              END_IF;  

              IF "APC".TI[6]> 3 AND NOT "DC".XT_HDL_SLID_BW THEN                    
                   #end_of_step := true;                            
              END_IF;                                      
                   #next_step := 220;

      //-----------------------------------------------------------                 
      // 22.step XT-Handling swivel drive to parking position 10?
      //-----------------------------------------------------------
      220:                                                           
              IF #next_step = #step THEN
                   #STEP_MSG  := 220;
                   "APC".TI[6] := 0;                                                  
              END_IF;

              IF "DIS".ACT_POS_XT_HDL_SW > 10.0 THEN
                 "DC".XT_HDL_SW_OUT   := TRUE;
                 ELSE
                 "DC".XT_HDL_SW_OUT  := FALSE;
              END_IF;

              IF "APC".TI[6]> 3 AND NOT "DC".XT_HDL_SW_OUT THEN                    
                  #end_of_step := true;                            
              END_IF;  
                  #next_step := 230;

      //-----------------------------------------------------------                 
      // 23.step XT-Handling lift drive in crystal position 2600 mm   
      //-----------------------------------------------------------
      230:                                                           
               IF #next_step = #step THEN
                   #STEP_MSG  := 230;
                   "APC".TI[6] := 0;                                                  
               END_IF;

               IF "DIS".ACT_POS_XT_HDL_LFT < 2600.0 THEN
                  "DC".XT_HDL_LFT_UP   := TRUE;                            
                  ELSE
                  "DC".XT_HDL_LFT_UP  := FALSE;
               END_IF;

                  "DC".XT_HDL_LFT_FAST := "DC".XT_HDL_LFT_UP AND "DIS".ACT_POS_XT_HDL_LFT >355.0;

               IF "DIS".ACT_POS_XT_HDL_LFT >= 2600.0 AND NOT "DC".XT_HDL_LFT_UP THEN   
                  "LT".XT_HDL_SEQ_XT_OUT := FALSE ;    // stop sub sequence
               END_IF;

               IF  "APC".TI[6]> 3 AND NOT "LT".XT_HDL_SEQ_XT_OUT THEN                    
                   #end_of_step := true;                            
               END_IF;   
                   #next_step := 0;   


      //-----------------------------------------------------------                 
      // Start sequencer Crucible handling
      // 1. step Check start conditions 
      //-----------------------------------------------------------
      300:                                                           
               IF #next_step = #step THEN
                   #STEP_MSG := 300;
                   "APC".TI[6] := 0; 
               END_IF; 

               "DC".XT_HDL_LFT_UP  := "DIS".ACT_POS_XT_HDL_LFT > 2500.0;    // 2500mm;      // Lift in upper safe position
               "DC".XT_HDL_SW_OUT  := "DIS".ACT_POS_XT_HDL_SW < 10.0;        // swivel drive in outer position
               "DC".XT_HDL_SLID_BW := NOT "PDI".LS_XT_SLID_BW;                   // slider drive in back position


               IF          "APC".TI[6]> 3 
                   AND NOT "DC".XT_HDL_LFT_UP 
                   AND NOT "DC".XT_HDL_SW_OUT 
                   AND NOT "DC".XT_HDL_SLID_BW 
                   AND     "PDI".LS_GCH_SW_OUT 
                   AND     "PDI".LS_TCH_SW_OUT 
                   AND     "AV".TEC_FLG_SW_ENC_POS >=167.0
                   AND     "AV".UP_FCH_SW_ENC_POS  >=167.0 
                   AND     "AV".LO_FCH_SW_ENC_POS >= 150.0 THEN 

                   #end_of_step := true;                            
               END_IF;   
                   #next_step := 320; 

      //--------------------------------------------------------------------------                 
      // 2.step CRU-Handling lift drive in HOI-TOOL installation position 350 mm
      //--------------------------------------------------------------------------
      320:                                                           
               IF #next_step = #step THEN
                   #STEP_MSG  := 320;
                   "APC".TI[6] := 0;                                                  
               END_IF;

               IF ABS("DIS".ACT_POS_XT_HDL_LFT-350.0)>1.0 THEN
                  "DC".XT_HDL_LFT_DN   := TRUE;
                  ELSE
                  "DC".XT_HDL_LFT_DN  := FALSE;
               END_IF;

                  "DC".XT_HDL_LFT_FAST := "DC".XT_HDL_LFT_DN AND "DIS".ACT_POS_XT_HDL_LFT <2495.0;

               IF "APC".TI[6]> 3 AND NOT "DC".XT_HDL_LFT_DN THEN                    
                   #end_of_step := true;                            
               END_IF;                                    
                   #next_step := 330; 


     //--------------------------------------------------------------------------                
     //  3.step CRU-Handling swivel-in drive in HOI-TOOL installation position 40?  Position noch zu definieren!!!
     //--------------------------------------------------------------------------
      330:                                                           
              IF #next_step = #step THEN
                   #STEP_MSG  := 330;
                   "APC".TI[6] := 0;                                                  
              END_IF;

              IF ABS("DIS".ACT_POS_XT_HDL_SW-40.0)>0.1 THEN
                 "DC".XT_HDL_SW_IN   := TRUE;
                 ELSE
                 "DC".XT_HDL_SW_IN  := FALSE;
              END_IF;

              IF "APC".TI[6]> 3 AND NOT "DC".XT_HDL_SW_IN THEN                    
                  #end_of_step := true;                            
              END_IF;                                    
                  #next_step := 340;


      //-----------------------------------------------------------                 
      // 4.step CRU-Handling HOI-TOOL installation and confirm 
      //-----------------------------------------------------------
      340:                                                           
               IF #next_step = #step THEN
                  #STEP_MSG  := 340;
                  "APC".TI[6] := 0;                                                  
               END_IF;

                  "LT".HOI_TOOL_INST  := TRUE;

               IF "PDI".LS_HOI_TOOL_INST THEN 
                  "LT".HOI_TOOL_INST := FALSE;
               END_IF;   

               IF "APC".TI[6]> 3 AND NOT "LT".HOI_TOOL_INST THEN                    
                  #end_of_step := true;                            
               END_IF;                                    
                  #next_step := 350;

      //-----------------------------------------------------------------------                 
      // 5.step CRU-Handling HOI-TOOL lift drive in takeover position 1000 mm   noch zu definieren!!! 
      //-----------------------------------------------------------------------
      350:                                                           
               IF #next_step = #step THEN
                   #STEP_MSG  := 350;
                   "APC".TI[6] := 0;                                                  
               END_IF;

               IF ABS("DIS".ACT_POS_XT_HDL_LFT - 1000.0) > 1.0 THEN
                  "DC".XT_HDL_LFT_UP   := TRUE;                            
                  ELSE
                  "DC".XT_HDL_LFT_UP  := FALSE;
               END_IF;

               "DC".XT_HDL_LFT_FAST := "DC".XT_HDL_LFT_UP AND "DIS".ACT_POS_XT_HDL_LFT >355.0;

               IF "APC".TI[6]> 3 AND NOT "DC".XT_HDL_LFT_UP THEN                    
                  #end_of_step := true;                            
               END_IF;                                    
                  #next_step := 360; 

      //------------------------------------------------------------------------                 
      // 6.step CRU-Handling HOI-TOOL swivel-in drive in takeover position 185?   Position noch zu definieren!!! 
      //------------------------------------------------------------------------
      360:                                                           
               IF #next_step = #step THEN
                  #STEP_MSG  := 360;
                  "APC".TI[6] := 0;                                                  
               END_IF;

                  "DC".XT_HDL_SW_IN := "DIS".ACT_POS_XT_HDL_SW < 185.0;

               IF "APC".TI[6]> 3 AND NOT "DC".XT_HDL_SW_IN THEN                    
                  #end_of_step := true;                            
               END_IF;                                        
                  #next_step := 370; 


      //-----------------------------------------------------------                 
      // 7.step CRU-Handling installation Crucible confirm  
      //-----------------------------------------------------------
     370:                                                           
               IF #next_step = #step THEN
                   #STEP_MSG  := 370;
                   "APC".TI[6] := 0;                                                  
               END_IF;

                  "LT".HOI_TOOL_CRU_INS := TRUE;

               IF "KYD".HOI_TOOL_CRU_INS THEN 
                   #end_of_step := true; 
                   "LT".HOI_TOOL_CRU_INS := FALSE;
                   "KYD".HOI_TOOL_CRU_INS:= FALSE;
               END_IF;    

               IF "APC".TI[6]> 3 AND NOT "LT".HOI_TOOL_CRU_INS THEN                    
                  #end_of_step := true;                            
               END_IF;                                      
                  #next_step := 380; 

      //-----------------------------------------------------------------------------------------                 
      // 8.step CRU-Handling HOI/TOOL with crucible swivel-out drive in transport car position 40? noch zu definieren!!
      //-----------------------------------------------------------------------------------------
      380:                                                           
              IF #next_step = #step THEN
                   #STEP_MSG  := 380;
                   "APC".TI[6] := 0;                                                  
              END_IF;

              IF ABS("DIS".ACT_POS_XT_HDL_SW - 40.0) > 1.0 THEN
                  "DC".XT_HDL_SW_OUT   := TRUE;                            
                  ELSE
                  "DC".XT_HDL_SW_OUT  := FALSE;
              END_IF;

              IF "APC".TI[6]> 3 AND NOT "DC".XT_HDL_SW_OUT THEN                    
                  #end_of_step := true;                            
              END_IF;                                    
                  #next_step := 390;

      //---------------------------------------------------------------------------------------------------------------------------------                 
      // 9.step CRU-Handling crucible from HOI/TOOL uninstallation and confirm crucible saftey on transport car/new crucible installation
      //---------------------------------------------------------------------------------------------------------------------------------
      390:                                                           
               IF #next_step = #step THEN
                   #STEP_MSG  := 390;  
                   "APC".TI[6] := 0;                                                  
               END_IF;

                  "LT".LD_CRU_OP_CONT := TRUE;
                  "LT".LD_CRU_FIN     := TRUE;

               IF "KYD".LD_CRU_OP_CONT AND NOT "KYD".LD_CRU_FIN THEN
                  #end_of_step := true; 
                  "LT".LD_CRU_OP_CONT := FALSE;
                  "LT".LD_CRU_FIN     := FALSE;
                  "KYD".LD_CRU_OP_CONT:= FALSE;
                  "KYD".LD_CRU_FIN    := FALSE; 
               END_IF;   

               IF "APC".TI[6]> 3 AND NOT "LT".LD_CRU_OP_CONT THEN                    
                  #end_of_step := true;                            
               END_IF;                                      
                  #next_step := 400; 


      //-----------------------------------------------------------------------------------                 
      // 10.step CRU-Handling HOI-TOOL with new CRU lift drive in CRU-install position 1000 mm   
      //-----------------------------------------------------------------------------------
      400:                                                           
               IF #next_step = #step THEN
                   #STEP_MSG  := 400;
                   "APC".TI[6] := 0;                                                  
               END_IF;

               IF ABS("DIS".ACT_POS_XT_HDL_LFT - 1000.0) > 1.0 THEN
                  "DC".XT_HDL_LFT_UP   := TRUE;                            
                  ELSE
                  "DC".XT_HDL_LFT_UP  := FALSE;
               END_IF;

             //  DC.XT_HDL_LFT_FAST := DC.XT_HDL_LFT_UP AND DIS.ACT_POS_XT_HDL_LFT >355.0;

               IF "APC".TI[6]> 3 AND NOT "DC".XT_HDL_LFT_UP THEN                    
                  #end_of_step := true;                            
               END_IF;                                    
                  #next_step := 410;


      //--------------------------------------------------------------------------------------                 
      // 11.step CRU-Handling HOI-TOOL with new CRU swivel-in drive in CRU-install position 185?                                      
      //--------------------------------------------------------------------------------------
      410:                                                           
               IF #next_step = #step THEN
                   #STEP_MSG  := 410;
                   "APC".TI[6] := 0;                                                  
               END_IF;

                  "DC".XT_HDL_SW_IN := "DIS".ACT_POS_XT_HDL_SW < 185.0 ; 

               IF "APC".TI[6]> 100 AND NOT "DC".XT_HDL_SW_IN THEN                    
                  #end_of_step := true;                            
               END_IF;                                    
                  #next_step := 420;

      //--------------------------------------------------------------------                 
      // 12.step CRU-Handling lift down in CRU saftey home position 800 mm        Position noch zu definieren!!  manually lift down ?? 
      //--------------------------------------------------------------------
      420:                                                           
               IF #next_step = #step THEN
                   #STEP_MSG  := 420;
                   "APC".TI[6] := 0;                                                  
               END_IF;

               IF ABS("DIS".ACT_POS_XT_HDL_LFT-800.0)>1.0 THEN
                  "DC".XT_HDL_LFT_DN   := TRUE;
                  ELSE
                  "DC".XT_HDL_LFT_DN  := FALSE;
               END_IF;

               IF "APC".TI[6]> 3 AND NOT "DC".XT_HDL_LFT_DN THEN                    
                  #end_of_step := true;                            
               END_IF;                                    
                  #next_step := 430; 


      //-----------------------------------------------------------                 
      // 13.step CRU-Handling HOI-TOOL lift up to position 1000 mm            
      //-----------------------------------------------------------
      430:                                                           

               IF #next_step = #step THEN
                   #STEP_MSG  := 430;
                   "APC".TI[6] := 0;                                                  
               END_IF;

               IF ABS("DIS".ACT_POS_XT_HDL_LFT-1000.0)>1.0 THEN
                  "DC".XT_HDL_LFT_UP   := TRUE;
                  ELSE
                  "DC".XT_HDL_LFT_UP   := FALSE;
               END_IF;

               IF "APC".TI[6]> 3 AND NOT "DC".XT_HDL_LFT_UP THEN                    
                  #end_of_step := true;                            
               END_IF;                                    
                  #next_step := 340; 


      //-------------------------------------------------------------------                 
      // 14.step CRU-Handling HOI-TOOL swivel out to uninstall position 40?       
      //-------------------------------------------------------------------
      440:                                                           
               IF #next_step = #step THEN
                   #STEP_MSG  := 440;
                   "APC".TI[6] := 0;                                                  
               END_IF;            

               IF ABS("DIS".ACT_POS_XT_HDL_SW - 40.0) > 1.0 THEN
                  "DC".XT_HDL_SW_OUT   := TRUE;                            
                  ELSE
                  "DC".XT_HDL_SW_OUT  := FALSE;
               END_IF;

               IF "APC".TI[6]> 3 AND NOT "DC".XT_CLP_TILT_75 THEN                    
                  #end_of_step := true;                            
               END_IF;                                   
                  #next_step := 450;

      //---------------------------------------------------------------------------------------------------------                 
      // 15.step CRU-Handling HOI-TOOL lift down to uninstall position 350mm and confirm if HOI-TOOL uninstalled       
      //---------------------------------------------------------------------------------------------------------
      450:                                                           
               IF #next_step = #step THEN
                   #STEP_MSG  := 450;
                   "APC".TI[6] := 0;                                                  
               END_IF;             

                  "LT".HOI_TOOL_UNIS := TRUE;

               IF "KYD".HOI_TOOL_UNIS AND NOT "PDI".LS_HOI_TOOL_INST THEN 

                  "LT".HOI_TOOL_UNIS := FALSE;
                  "KYD".HOI_TOOL_UNIS:= FALSE;

               END_IF;

               IF "APC".TI[6]> 3 AND NOT "LT".HOI_TOOL_UNIS THEN 
                   #end_of_step := true;                            
               END_IF;                                   
                   #next_step := 460;

      //-----------------------------------------------------------                 
      // 16.step CRU-Handling Handling-arm drive to home position 10?    
      //-----------------------------------------------------------
      460:                                                           
               IF #next_step = #step THEN
                   #STEP_MSG  := 460;
                   "APC".TI[6] := 0;                                                  
               END_IF;

                   "DC".XT_HDL_SW_OUT := "DIS".ACT_POS_XT_HDL_SW > 10.0;

               IF "APC".TI[6]> 3 AND NOT "DC".XT_HDL_SW_OUT THEN                    
                  #end_of_step := true;                            
               END_IF;                                    
                  #next_step := 470;

      //----------------------------------------------------------------                 
      // 17.step CRU-Handling Handling-arm drive to home position 2500mm        
      //----------------------------------------------------------------
      470:                                                           
               IF #next_step = #step THEN
                   #STEP_MSG  := 470;
                   "APC".TI[6] := 0;                                                  
               END_IF;

                  "DC".XT_HDL_LFT_UP   := "DIS".ACT_POS_XT_HDL_LFT < 2500.0; 
                  "DC".XT_HDL_LFT_FAST := "DC".XT_HDL_LFT_UP AND "DIS".ACT_POS_XT_HDL_LFT >355.0;

               IF "APC".TI[6]> 3 AND NOT "DC".XT_HDL_LFT_UP THEN                    
                  #end_of_step := true;                            
               END_IF;  


               IF "DIS".ACT_POS_XT_HDL_LFT >= 2600.0 AND NOT "DC".XT_HDL_LFT_UP THEN   
                  "LT".XT_HDL_SEQ_LD_CRU := FALSE ;  // stop sub sequence CRU-Handling
               END_IF;

               IF  "APC".TI[6]> 3 AND NOT "LT".XT_HDL_SEQ_LD_CRU THEN                    
                   #end_of_step := true;                            
               END_IF;   
                   #next_step := 0;   



      //-----------------------------------------------------------                 
      // Start sequencer Hotzone handling
      // 1. step Check start conditions 
      //-----------------------------------------------------------
      600:                                                               
               IF #next_step = #step THEN
                   #STEP_MSG := 600;
                   "APC".TI[6] := 0; 
               END_IF; 

               "DC".XT_HDL_LFT_UP  := "DIS".ACT_POS_XT_HDL_LFT > 2500.0;    // 2500mm;      // Lift in upper safe position
               "DC".XT_HDL_SW_OUT  := "DIS".ACT_POS_XT_HDL_SW < 10.0;       // swivel drive in outer position
               "DC".XT_HDL_SLID_BW := NOT "PDI".LS_XT_SLID_BW;              // slider drive in back position

               IF          "APC".TI[6]> 3 
                   AND NOT "DC".XT_HDL_LFT_UP 
                   AND NOT "DC".XT_HDL_SW_OUT 
                   AND NOT "DC".XT_HDL_SLID_BW 
                   AND     "PDI".LS_GCH_SW_OUT 
                   AND     "PDI".LS_TCH_SW_OUT 
                   AND     "AV".TEC_FLG_SW_ENC_POS >=167.0
                   AND     "AV".UP_FCH_SW_ENC_POS  >=167.0 
                   AND     "AV".LO_FCH_SW_ENC_POS >= 150.0 THEN 

                   #end_of_step := true;                            
               END_IF;   
                   #next_step := 620; 

      //--------------------------------------------------------------------------                 
      // 2.step Hotzone Handling lift drive in HOI-TOOL installation position 350 mm
      //--------------------------------------------------------------------------
      620:                                                        
               IF #next_step = #step THEN
                   #STEP_MSG  := 620;
                   "APC".TI[6] := 0;                                                  
               END_IF;

               IF ABS("DIS".ACT_POS_XT_HDL_LFT-350.0)>1.0 THEN
                  "DC".XT_HDL_LFT_DN   := TRUE;
                  ELSE
                  "DC".XT_HDL_LFT_DN  := FALSE;
               END_IF;

                  "DC".XT_HDL_LFT_FAST := "DC".XT_HDL_LFT_DN AND "DIS".ACT_POS_XT_HDL_LFT <2495.0;

               IF "APC".TI[6]> 3 AND NOT "DC".XT_HDL_LFT_DN THEN                    
                   #end_of_step := true;                            
               END_IF;                                    
                   #next_step := 630; 


     //--------------------------------------------------------------------------                
     //  3.step Hotzone Handling swivel-in drive in HOI-TOOL installation position 40?  Position noch zu definieren!!!
     //--------------------------------------------------------------------------
      630:                                                           
              IF #next_step = #step THEN
                   #STEP_MSG  := 630;
                   "APC".TI[6] := 0;                                                  
              END_IF;

              IF ABS("DIS".ACT_POS_XT_HDL_SW-40.0)>0.1 THEN
                 "DC".XT_HDL_SW_IN   := TRUE;
                 ELSE
                 "DC".XT_HDL_SW_IN  := FALSE;
              END_IF;

              IF "APC".TI[6]> 3 AND NOT "DC".XT_HDL_SW_IN THEN                    
                  #end_of_step := true;                            
              END_IF;                                    
                  #next_step := 640;


      //-----------------------------------------------------------                 
      // 4.step Hotzone Handling HOI-TOOL installation and confirm 
      //-----------------------------------------------------------
      640:                                                           
               IF #next_step = #step THEN
                  #STEP_MSG  := 640;
                  "APC".TI[6] := 0;                                                  
               END_IF;

                  "LT".HOI_TOOL_INST  := TRUE;

               IF "PDI".LS_HOI_TOOL_INST THEN 
                  "LT".HOI_TOOL_INST := FALSE;
               END_IF;   

               IF "APC".TI[6]> 3 AND NOT "LT".HOI_TOOL_INST THEN                    
                  #end_of_step := true;                            
               END_IF;                                    
                  #next_step := 650;

      //-----------------------------------------------------------------------                 
      // 5.step Hotzone Handling HOI-TOOL lift drive in takeover position 1000 mm   noch zu definieren!!! 
      //-----------------------------------------------------------------------
      650:                                                           
               IF #next_step = #step THEN
                   #STEP_MSG  := 650;
                   "APC".TI[6] := 0;                                                  
               END_IF;

               IF ABS("DIS".ACT_POS_XT_HDL_LFT - 1000.0) > 1.0 THEN
                  "DC".XT_HDL_LFT_UP   := TRUE;                            
                  ELSE
                  "DC".XT_HDL_LFT_UP  := FALSE;
               END_IF;

               "DC".XT_HDL_LFT_FAST := "DC".XT_HDL_LFT_UP AND "DIS".ACT_POS_XT_HDL_LFT >355.0;

               IF "APC".TI[6]> 3 AND NOT "DC".XT_HDL_LFT_UP THEN                    
                  #end_of_step := true;                            
               END_IF;                                    
                  #next_step := 660; 

      //------------------------------------------------------------------------                 
      // 6.step Hotzone Handling HOI-TOOL swivel-in drive in takeover position 185?   Position noch zu definieren!!! 
      //------------------------------------------------------------------------
      660:                                                           
               IF #next_step = #step THEN
                  #STEP_MSG  := 660;
                  "APC".TI[6] := 0;                                                  
               END_IF;

                  "DC".XT_HDL_SW_IN := "DIS".ACT_POS_XT_HDL_SW < 185.0;

               IF "APC".TI[6]> 3 AND NOT "DC".XT_HDL_SW_IN THEN                    
                  #end_of_step := true;                            
               END_IF;                                        
                  #next_step := 670; 


      //-----------------------------------------------------------                 
      // 7.step Hotzone Handling installation Hotzone and confirm it  
      //-----------------------------------------------------------
     670:                                                           
               IF #next_step = #step THEN
                   #STEP_MSG  := 670;
                   "APC".TI[6] := 0;                                                  
               END_IF;

                  "LT".HOI_TOOL_HZ_INS := TRUE;

               IF "KYD".HOI_TOOL_HZ_INS THEN 
                   #end_of_step := true; 
                   "LT".HOI_TOOL_HZ_INS := FALSE;
                   "KYD".HOI_TOOL_HZ_INS:= FALSE;
               END_IF;    

               IF "APC".TI[6]> 3 AND NOT "LT".HOI_TOOL_HZ_INS THEN                    
                  #end_of_step := true;                            
               END_IF;                                      
                  #next_step := 680; 

      //---------------------------------------------------------------------------------------------                
      // 8.step Hotzone Handling HOI/TOOL with Hotzone swivel-out drive in transport car position 40? noch zu definieren!!
      //---------------------------------------------------------------------------------------------
      680:                                                           
              IF #next_step = #step THEN
                   #STEP_MSG  := 680;
                   "APC".TI[6] := 0;                                                  
              END_IF;

              IF ABS("DIS".ACT_POS_XT_HDL_SW - 40.0) > 1.0 THEN
                  "DC".XT_HDL_SW_OUT   := TRUE;                            
                  ELSE
                  "DC".XT_HDL_SW_OUT  := FALSE;
              END_IF;

              IF "APC".TI[6]> 3 AND NOT "DC".XT_HDL_SW_OUT THEN                    
                  #end_of_step := true;                            
              END_IF;                                    
                  #next_step := 690;

      //---------------------------------------------------------------------------------------------------------------------------------                 
      // 9.step Hotzone Handling Hotzone from HOI/TOOL uninstallation and confirm Hotzone saftey on transport car/new Hotzone installation
      //---------------------------------------------------------------------------------------------------------------------------------
      690:                                                           
               IF #next_step = #step THEN
                   #STEP_MSG  := 690;  
                   "APC".TI[6] := 0;                                                  
               END_IF;

                  "LT".LD_HZ_OP_CONT := TRUE;
                  "LT".LD_HZ_FIN     := TRUE;

               IF "KYD".LD_HZ_OP_CONT AND NOT "KYD".LD_HZ_FIN THEN
                  #end_of_step := true; 
                  "LT".LD_HZ_OP_CONT := FALSE;
                  "LT".LD_HZ_FIN     := FALSE;
                  "KYD".LD_HZ_OP_CONT:= FALSE;
                  "KYD".LD_HZ_FIN    := FALSE; 
               END_IF;   

               IF "APC".TI[6]> 3 AND NOT "LT".LD_HZ_OP_CONT THEN                    
                  #end_of_step := true;                            
               END_IF;                                      
                  #next_step := 700; 

      //--------------------------------------------------------------------------------------------------                 
      // 10.step Hotzone Handling HOI-TOOL with new Hotzone lift drive in Hotzone-Install position 1000 mm   
      //--------------------------------------------------------------------------------------------------
      700:                                                           
               IF #next_step = #step THEN
                   #STEP_MSG  := 700; 
                   "APC".TI[6] := 0;                                                  
               END_IF;

               IF ABS("DIS".ACT_POS_XT_HDL_LFT - 1000.0) > 1.0 THEN
                  "DC".XT_HDL_LFT_UP   := TRUE;                            
                  ELSE
                  "DC".XT_HDL_LFT_UP  := FALSE;
               END_IF;

             //  DC.XT_HDL_LFT_FAST := DC.XT_HDL_LFT_UP AND DIS.ACT_POS_XT_HDL_LFT >355.0;

               IF "APC".TI[6]> 3 AND NOT "DC".XT_HDL_LFT_UP THEN                    
                  #end_of_step := true;                            
               END_IF;                                    
                  #next_step := 710;


      //-----------------------------------------------------------------------------------------------------                 
      // 11.step Hotzone Handling HOI-TOOL with new Hotzone swivel-in drive in Hotzone-Install position 185?                                      
      //-----------------------------------------------------------------------------------------------------
      710:                                                           
               IF #next_step = #step THEN
                   #STEP_MSG  := 710;
                   "APC".TI[6] := 0;                                                  
               END_IF;

                  "DC".XT_HDL_SW_IN := "DIS".ACT_POS_XT_HDL_SW < 185.0 ; 

               IF "APC".TI[6]> 100 AND NOT "DC".XT_HDL_SW_IN THEN                    
                  #end_of_step := true;                            
               END_IF;                                    
                  #next_step := 720;

      //--------------------------------------------------------------------------                 
      // 12.step Hotzone Handling lift down in Hotzone saftey home position 800 mm        Position noch zu definieren!!  manually lift down ?? 
      //--------------------------------------------------------------------------
      720:                                                           
               IF #next_step = #step THEN
                   #STEP_MSG  := 720;
                   "APC".TI[6] := 0;                                                  
               END_IF;

               IF ABS("DIS".ACT_POS_XT_HDL_LFT-800.0)>1.0 THEN
                  "DC".XT_HDL_LFT_DN   := TRUE;
                  ELSE
                  "DC".XT_HDL_LFT_DN  := FALSE;
               END_IF;

               IF "APC".TI[6]> 3 AND NOT "DC".XT_HDL_LFT_DN THEN                    
                  #end_of_step := true;                            
               END_IF;                                    
                  #next_step := 730; 

      //-----------------------------------------------------------                 
      // 13.step Hotzone Handling HOI-TOOL lift up to position 1000 mm            
      //-----------------------------------------------------------
      730:                                                           

               IF #next_step = #step THEN
                   #STEP_MSG  := 730;
                   "APC".TI[6] := 0;                                                  
               END_IF;

               IF ABS("DIS".ACT_POS_XT_HDL_LFT-1000.0)>1.0 THEN
                  "DC".XT_HDL_LFT_UP   := TRUE;
                  ELSE
                  "DC".XT_HDL_LFT_UP   := FALSE;
               END_IF;

               IF "APC".TI[6]> 3 AND NOT "DC".XT_HDL_LFT_UP THEN                    
                  #end_of_step := true;                            
               END_IF;                                    
                  #next_step := 740; 


      //-------------------------------------------------------------------                 
      // 17.step Hotzone Handling HOI-TOOL swivel out to uninstall position 40?       
      //-------------------------------------------------------------------
      740:                                                           
               IF #next_step = #step THEN
                   #STEP_MSG  := 740;
                   "APC".TI[6] := 0;                                                  
               END_IF;            

               IF ABS("DIS".ACT_POS_XT_HDL_SW - 40.0) > 1.0 THEN
                  "DC".XT_HDL_SW_OUT   := TRUE;                            
                  ELSE
                  "DC".XT_HDL_SW_OUT  := FALSE;
               END_IF;

               IF "APC".TI[6]> 3 AND NOT "DC".XT_CLP_TILT_75 THEN                    
                  #end_of_step := true;                            
               END_IF;                                   
                  #next_step := 750;

      //--------------------------------------------------------------------------------------------------------------                 
      // 15.step Hotzone Handling HOI-TOOL lift down to uninstall position 350mm and confirm if HOI-TOOL uninstalled       
      //--------------------------------------------------------------------------------------------------------------
      750:                                                           
               IF #next_step = #step THEN
                   #STEP_MSG  := 750;
                   "APC".TI[6] := 0;                                                  
               END_IF;             

                  "LT".HOI_TOOL_UNIS := TRUE;

               IF "KYD".HOI_TOOL_UNIS AND NOT "PDI".LS_HOI_TOOL_INST THEN 

                  "LT".HOI_TOOL_UNIS := FALSE;
                  "KYD".HOI_TOOL_UNIS:= FALSE;

               END_IF;

               IF "APC".TI[6]> 3 AND NOT "LT".HOI_TOOL_UNIS THEN 
                   #end_of_step := true;                            
               END_IF;                                   
                   #next_step := 760;

      //-----------------------------------------------------------------                 
      // 16.step Hotzone Handling Handling-arm drive to home position 10?    
      //-----------------------------------------------------------------
      760:                                                           
               IF #next_step = #step THEN
                   #STEP_MSG  := 760;
                   "APC".TI[6] := 0;                                                  
               END_IF;

                   "DC".XT_HDL_SW_OUT := "DIS".ACT_POS_XT_HDL_SW > 10.0;

               IF "APC".TI[6]> 3 AND NOT "DC".XT_HDL_SW_OUT THEN                    
                  #end_of_step := true;                            
               END_IF;                                    
                  #next_step := 770;

      //--------------------------------------------------------------------                 
      // 17.step Hotzone Handling Handling-arm drive to home position 2500mm        
      //--------------------------------------------------------------------
      770:                                                           
               IF #next_step = #step THEN
                   #STEP_MSG  := 770;
                   "APC".TI[6] := 0;                                                  
               END_IF;

                  "DC".XT_HDL_LFT_UP := "DIS".ACT_POS_XT_HDL_LFT < 2500.0; 
                  "DC".XT_HDL_LFT_FAST := "DC".XT_HDL_LFT_UP AND "DIS".ACT_POS_XT_HDL_LFT >355.0;

               IF "APC".TI[6]> 3 AND NOT "DC".XT_HDL_LFT_UP THEN                    
                  #end_of_step := true;                            
               END_IF;  


               IF "DIS".ACT_POS_XT_HDL_LFT >= 2600.0 AND NOT "DC".XT_HDL_LFT_UP THEN   
                  "LT".XT_HDL_SEQ_HDL_HZ := FALSE ;         // stop sub sequence Hotzone-Handling
               END_IF;

               IF  "APC".TI[6]> 3 AND NOT "LT".XT_HDL_SEQ_HDL_HZ THEN                    
                   #end_of_step := true;                            
               END_IF;   
                   #next_step := 0;          

       END_CASE;

              IF #end_of_step  AND (#step<1000) THEN
                  #step := #next_step; 
                  #end_of_step := False;      
              END_IF;
END_FUNCTION_BLOCK

FUNCTION_BLOCK "BM_VSL_HDL"   // FB62, SCL
{ S7_Optimized_Access := 'FALSE' }
VERSION : 0.0
// --------------------------------------------------------------------------------
//     program     :   BM_VSL_HDL
//     description :   handling of vessel parts
//     name        :   John Wang
//     date        :   08.11.2018
//   
//     revision    :
//     name        :
//     date        :    
//                     (c)PVA CGS GmbH
//     --------------------------------------------------------------------------------
   VAR
      BEL_LFT : "PM_DRV_COMM_LZI550";
      GCH_LFT : "PM_DRV_COMM_LZI550";
      TCH_LFT : "PM_DRV_COMM_LZI550";
      TCH_TILT : "PM_DRV_COMM_LZI550";
      TEC_FLG_LFT : "PM_DRV_COMM_LZI550";
      FCH_LFT : "PM_DRV_COMM_LZI550";
      V7_LFT : "PM_DRV_COMM_LZI550";
      V7_SW : "PM_DRV_COMM_LZI550";
      DELAY_MAG_DRV_ON : S5Time := S5T#2S;   // magnet drive start delay
      BI_TMR_MAG_DRV : Word;
      DELAY_FCH_SW_BRK_OFF : Int := 3;
      BI_TMR_TEC_FLG_SW : Int;
      BI_TMR_UP_FCH_SW : Int;
      BI_TMR_LO_FCH_SW : Int;
      mag_drv_dly_over : Bool;
      tec_flg_sw_unlock : Bool;
      up_fch_sw_unlock : Bool;
      lo_fch_sw_unlock : Bool;
      auto_gch_sw_lock : Bool;
      fl_gch_sw_lock : Bool;
      auto_tch_sw_lock : Bool;
      fl_tch_sw_lock : Bool;
      kyd_up_fch_unlock : Bool;
      BEL_LFT_FU_RDY : Bool;
      BEL_LFT_SPD_RCH : Bool;
      BEL_LFT_RUN : Bool;
      BEL_ERROR_CODE : DInt;
      BEL_ACT_SETP : Real;
      GCH_LFT_FU_RDY : Bool;
      GCH_LFT_SPD_RCH : Bool;
      GCH_LFT_RUN : Bool;
      GCH_ERROR_CODE : DInt;
      GCH_ACT_SETP : Real;
      V7_LFT_FU_RDY : Bool;
      V7_LFT_SPD_RCH : Bool;
      V7_LFT_RUN : Bool;
      V7_LFT_ERROR_CODE : DInt;
      V7_LFT_ACT_SETP : Real;
      V7_SW_FU_RDY : Bool;
      V7_SW_SPD_RCH : Bool;
      V7_SW_RUN : Bool;
      V7_SW_ERROR_CODE : DInt;
      V7_SW_ACT_SETP : Real;
      TCH_LFT_FU_RDY : Bool;
      TCH_LFT_SPD_RCH : Bool;
      TCH_LFT_RUN : Bool;
      TCH_LFT_ERROR_CODE : DInt;
      TCH_LFT_ACT_SETP : Real;
      TCH_TILT_FU_RDY : Bool;
      TCH_TILT_SPD_RCH : Bool;
      TCH_TILT_RUN : Bool;
      TCH_TILT_ERROR_CODE : DInt;
      TCH_TILT_ACT_SETP : Real;
      TEC_FLG_LFT_FU_RDY : Bool;
      TEC_FLG_LFT_SPD_RCH : Bool;
      TEC_FLG_LFT_RUN : Bool;
      TEC_FLG_LFT_ERROR_CODE : DInt;
      TEC_FLG_LFT_ACT_SETP : Real;
      FCH_LFT_FU_RDY : Bool;
      FCH_LFT_SPD_RCH : Bool;
      FCH_LFT_RUN : Bool;
      FCH_LFT_ERROR_CODE : DInt;
      FCH_LFT_ACT_SETP : Real;
      OLD_TEC_FLG_SW_POS : Real;
      OLD_UP_FCH_SW_POS : Real;
      OLD_LO_FCH_SW_POS : Real;
      TEC_FLG_SET_SPD : Real;
      FCH_LFT_SET_SPD : Real;
      mag_pos_cal : Real;
   END_VAR
   VAR_TEMP
      iTime : S5Time;   // Returnvalue function S_ODT
      diff_prs_ok : Bool;
      rel_drv_xt_pos : Bool;
   END_VAR
BEGIN

      "DV".MP_SERVICE := "KYD".KEY_PROCESS  AND ("STA".ACT_STATE = 2);
      "LT".MP_SERVICE := "DV".MP_SERVICE;

      "PDO".FU_FCB_HDL_ON := "PDI".EMO;
      "PDO".FU_GCB_HDL_ON := "PDI".EMO;


      //----------------------------------------------------------------------
      // bellow lift drive
      //----------------------------------------------------------------------
      // bellow lift up   
      "CM_ITL_IO"(ADR := 40,
             KYD_ON := "KYD".BEL_LFT_UP AND "PDI".MP_ENB_K9,
             KYD_OFF := NOT "KYD".BEL_LFT_UP OR NOT "PDI".MP_ENB_K9,
             AUTO := "APC".AUTOMATIC, 
             DC_ON := "SysLog0",
             CON1 := "PDI".EMO AND "PDI".EMS,
             CON2 := NOT "FLT".BEL_LFT_ERR,                    
             CON3 := NOT "LT".BEL_LFT_DN,
             CON4 := "DV".APS_GCH_DELAYED OR "DV".MP_SERVICE,
             CON5 := "PDI".LS_GCH_BEL_UP,                       
             CON6 := "DIS".ACT_XT_POS < "CNF".xt_high_pos + 5.0,    
             CON7 := "SysLog1",   
             CON8 := "SysLog1",   
             ITL_OUT := "STA_ITL_CAUSE",
             LT_OUT := "LT".BEL_LFT_UP); 

      "LT".BEL_LFT_UP_REL :=         "PDI".EMO AND "PDI".EMS 
                           AND NOT "FLT".BEL_LFT_ERR 
                           AND     "PDI".LS_GCH_BEL_UP
                           AND     "DV".APS_GCH_DELAYED
                           AND NOT "LT".BEL_LFT_DN 
                           AND     "DIS".ACT_XT_POS < "CNF".xt_high_pos + 5.0; 

      // bellow lift down   
      "CM_ITL_IO"(ADR := 41,
             KYD_ON := "KYD".BEL_LFT_DN  AND "PDI".MP_ENB_K9,
             KYD_OFF := NOT "KYD".BEL_LFT_DN  OR NOT "PDI".MP_ENB_K9,
             AUTO := "APC".AUTOMATIC,
             DC_ON:= "SysLog0",
             CON1 := "PDI".EMO AND "PDI".EMS,
             CON2 := NOT "FLT".BEL_LFT_ERR,                    
             CON3 := NOT "LT".BEL_LFT_UP,
             CON4 := ("PDI".LS_GCH_SW_IN AND "PDI".LS_GCH_DN) OR ("PDI".LS_GCH_SW_OUT AND "DV".MP_SERVICE),
             CON5 := "SysLog1",   
             CON6 := "PDI".LS_GCH_BEL_DN,   
             CON7 := "SysLog1",    
             CON8 := "SysLog1",   
             ITL_OUT:= "STA_ITL_CAUSE",
             LT_OUT := "LT".BEL_LFT_DN);

      "LT".BEL_LFT_DN_REL :=         "PDI".EMO AND "PDI".EMS 
                           AND NOT "FLT".BEL_LFT_ERR
                           AND   (("PDI".LS_GCH_SW_IN AND "PDI".LS_GCH_DN) OR ("PDI".LS_GCH_SW_OUT AND "DV".MP_SERVICE))
                           AND     "PDI".LS_GCH_BEL_DN
                           AND NOT "LT".BEL_LFT_UP;

      IF "CNF_BEL_LFT_LZ550".CTRL_ACTIV = 1 THEN 

           "PDO".BEL_LFT_ENB   :=  True;  // controller enable bellow lift





         #BEL_LFT(Enable         := "LT".BEL_LFT_UP OR "LT".BEL_LFT_DN, 
                   CW              := "LT".BEL_LFT_UP,   //  lift up
                   CCW             := "LT".BEL_LFT_DN,   //  lift down
                   Stopp           := NOT "LT".BEL_LFT_UP AND NOT "LT".BEL_LFT_DN,
                   Reset_error     := "KYD".BEL_LFT_TRIP_RES,
                   Speed_Hz        := "CNF_BEL_LFT_LZ550".SETP,
                   PM_ADR_E        := INT_TO_WORD ("CNF_BEL_LFT_LZ550".PE_ADR),
                   PM_ADR_A        := INT_TO_WORD ("CNF_BEL_LFT_LZ550".PA_ADR)); 


        "FLT".BEL_LFT_ERR     :=  #BEL_LFT.Error;
       // BEL_LFT_FU_RDY      :=  BEL_LFT.READY OR SY.SIM_ON;  
        #BEL_LFT_SPD_RCH     :=  #BEL_LFT.Speed_reached;
      //  BEL_LFT_RUN         :=  BEL_LFT.RUNNING;    
        #BEL_ERROR_CODE      :=  #BEL_LFT.Error_code;
        #BEL_ACT_SETP        :=  #BEL_LFT.Act_Speed_Hz;

       END_IF;


      //----------------------------------------------------------------------
      //Gate chamber lift drive
      //----------------------------------------------------------------------
      // Gate chamber lift up   
      "CM_ITL_IO"(ADR := 42,                                
             KYD_ON := "KYD".GCH_LFT_UP AND "PDI".MP_ENB_K9,
             KYD_OFF := NOT "KYD".GCH_LFT_UP OR NOT "PDI".MP_ENB_K9,
             AUTO := "APC".AUTOMATIC,
             DC_ON := "SysLog0",
             CON1 := "PDI".EMO AND "PDI".EMS,
             CON2 := NOT "FLT".GCH_LFT_ERR, 
             CON3 := NOT "LT".GCH_LFT_DN, 
             CON4 := "PDI".SLS_GCH_LFT AND "DV".APS_FCH_DELAYED AND "DV".V9_2_DLY_OP,   
             CON5 := NOT "PDI".LS_GCH_BEL_UP AND "PDI".LS_GCH_BEL_DN, 
             CON6 := "PDI".LS_TCH_DN AND "PDI".LS_TCH_SW_IN, 
             CON7 := NOT "PDI".LS_GCH_UP,                    
             CON8 := "PDI".LS_GCH_SW_IN AND "PDI".LS_GCH_DOOR_CL,       
             ITL_OUT := "STA_ITL_CAUSE",
             LT_OUT := "LT".GCH_LFT_UP);


       "LT".GCH_LFT_UP_REL :=     "PDI".EMO AND "PDI".EMS 
                            AND NOT "FLT".GCH_LFT_ERR
                            AND NOT "LT".GCH_LFT_DN
                            AND "PDI".SLS_GCH_LFT AND "DV".APS_FCH_DELAYED AND "DV".V9_2_DLY_OP   
                            AND NOT "PDI".LS_GCH_BEL_UP AND "PDI".LS_GCH_BEL_DN 
                            AND "PDI".LS_TCH_DN AND "PDI".LS_TCH_SW_IN  
                            AND NOT "PDI".LS_GCH_UP 
                            AND "PDI".LS_GCH_SW_IN AND "PDI".LS_GCH_DOOR_CL;    

       // gate chamber lift down

       "CM_ITL_IO"(ADR := 43,                                
             KYD_ON := "KYD".GCH_LFT_DN AND "PDI".MP_ENB_K9,
             KYD_OFF := NOT "KYD".GCH_LFT_DN  OR NOT "PDI".MP_ENB_K9,
             AUTO := "APC".AUTOMATIC,
             DC_ON := "SysLog0",
             CON1 := "PDI".EMO AND "PDI".EMS,
             CON2 := NOT "FLT".GCH_LFT_ERR, 
             CON3 := NOT "LT".GCH_LFT_UP,  
             CON4 := "PDI".LS_TCH_DN,
             CON5 := NOT "PDI".LS_GCH_DN,   
             CON6 := "PDI".LS_GCH_SW_IN,    
             CON7 := "PDI".SLS_GCH_LFT,   
             CON8 := "PDI".LS_TCH_SW_IN AND "PDI".LS_GCH_DOOR_CL,   
             ITL_OUT:= "STA_ITL_CAUSE",
             LT_OUT := "LT".GCH_LFT_DN);


       "LT".GCH_LFT_DN_REL :=    "PDI".EMO AND "PDI".EMS 
                           AND NOT "FLT".GCH_LFT_ERR 
                           AND NOT "LT".GCH_LFT_UP
                           AND "PDI".LS_TCH_DN   
                           AND NOT "PDI".LS_GCH_DN
                           AND "PDI".LS_GCH_SW_IN
                           AND "PDI".SLS_GCH_LFT
                           AND "PDI".LS_TCH_SW_IN AND "PDI".LS_GCH_DOOR_CL;   

       IF   "CNF_GCH_LFT_LZ550".CTRL_ACTIV=1 THEN 

             "PDO".GCH_LFT_ENB   :=  true;

          #GCH_LFT  (Enable         := "LT".GCH_LFT_UP OR "LT".GCH_LFT_DN, 
                   CW              := "LT".GCH_LFT_UP,   //  lift up
                   CCW             := "LT".GCH_LFT_DN,   //  lift down
                   Stopp           := NOT "LT".GCH_LFT_UP AND NOT "LT".GCH_LFT_DN,
                   Reset_error     := "KYD".CGT_LFT_TRIP_RES,
                   Speed_Hz        := "CNF_GCH_LFT_LZ550".SETP,
                   PM_ADR_E        := INT_TO_WORD ("CNF_GCH_LFT_LZ550".PE_ADR),
                   PM_ADR_A        := INT_TO_WORD ("CNF_GCH_LFT_LZ550".PA_ADR)); 



        "FLT".GCH_LFT_ERR     :=  #GCH_LFT.Error;
        #GCH_LFT_FU_RDY      :=  #GCH_LFT.Ready OR "SY".SIM_ON;  
        #GCH_LFT_SPD_RCH     :=  #GCH_LFT.Speed_reached;
        #GCH_LFT_RUN         :=  #GCH_LFT.Running;    
        #GCH_ERROR_CODE      :=  #GCH_LFT.Error_code;
        #GCH_ACT_SETP        :=  #GCH_LFT.Act_Speed_Hz;   

        END_IF; 


      // gate chamber swivel in / out release
      //----------------------------------------------------------------------
       "CM_ITL_IO"(ADR := 44,                                
             KYD_ON := "KYD".GCH_SW_UNLOCK AND "PDI".MP_ENB_K9,
             KYD_OFF := NOT "KYD".GCH_SW_UNLOCK OR NOT "PDI".MP_ENB_K9,
             AUTO := "APC".AUTOMATIC,
             DC_ON := "SysLog0",
             CON1 := "PDI".EMO AND "PDI".EMS,
             CON2 := NOT "PDI".LS_GCH_BEL_UP,
             CON3 := "PDI".LS_GCH_UP,
             CON4 := "PDI".LS_TCH_DN AND "PDI".LS_TCH_SW_IN,
             CON5 := "PDI".LS_TEC_FLG_DN, 
             CON6 := NOT "PDO".GCH_SW_LOCK,
             CON7 := "SysLog1",    
             CON8 := "SysLog1",   
             ITL_OUT:= "STA_ITL_CAUSE",
             LT_OUT := "PDO".GCH_SW_UNLOCK);


       "CM_ITL_IO"(ADR := 39,                                
             KYD_ON := ("KYD".GCH_SW_LOCK AND "PDI".MP_ENB_K9) OR #auto_gch_sw_lock,
             KYD_OFF := (NOT "KYD".GCH_SW_LOCK OR NOT "PDI".MP_ENB_K9) AND NOT #auto_gch_sw_lock,
             AUTO := "APC".AUTOMATIC,
             DC_ON := "SysLog0",
             CON1 := "PDI".EMO AND "PDI".EMS,
             CON2 := NOT "PDI".LS_GCH_BEL_UP,
             CON3 := "PDI".LS_GCH_UP,
             CON4 := "PDI".LS_TCH_DN AND "PDI".LS_TCH_SW_IN,
             CON5 := "PDI".LS_TEC_FLG_DN, 
             CON6 := NOT "PDO".GCH_SW_UNLOCK,
             CON7 := "PDI".LS_GCH_SW_IN OR "PDI".LS_GCH_SW_OUT OR "PDI".LS_GCH_SW_CLN,    
             CON8 := "SysLog1",   
             ITL_OUT:= "STA_ITL_CAUSE",
             LT_OUT := "PDO".GCH_SW_LOCK);

      IF ("PDI".LS_GCH_SW_IN OR "PDI".LS_GCH_SW_OUT) AND NOT #fl_gch_sw_lock THEN 
         #auto_gch_sw_lock := TRUE; 
         #fl_gch_sw_lock   := TRUE;                
      ELSE
         IF #auto_gch_sw_lock AND "PDI".LS_GCH_SW_LOCK THEN
            #auto_gch_sw_lock := FALSE;
         END_IF;
         IF NOT "PDI".LS_GCH_SW_IN AND NOT "PDI".LS_GCH_SW_OUT THEN
            #fl_gch_sw_lock   :=  FALSE;
         END_IF;
      END_IF;

      "LT".GCH_SW_OUT_REL   :=  NOT "PDI".LS_GCH_BEL_UP AND "PDI".LS_GCH_UP AND "PDI".LS_TCH_DN AND "PDI".LS_TCH_SW_IN AND "PDI".LS_TEC_FLG_DN AND
                              ("PDI".LS_GCH_SW_IN OR "PDI".LS_GCH_SW_OUT OR "PDI".LS_GCH_SW_CLN); 
      "LT".GCH_SW_IN_REL    :=  "LT".GCH_SW_OUT_REL;

      //  gate chamber light signal unlock
      "LT".GCH_SW_UNLOCK   := NOT "PDI".LS_GCH_SW_LOCK AND NOT "PDO".GCH_SW_LOCK AND NOT "PDO".GCH_SW_UNLOCK;
      "LT".GCH_SW_LOCKED   := "PDI".LS_GCH_SW_LOCK;

      //----------------------------------------------------------------------
      //Top chamber lift drive
      //----------------------------------------------------------------------
      // top chamber lift up   
      "CM_ITL_IO"(ADR := 45,                                
             KYD_ON := "KYD".TCH_LFT_UP AND "PDI".MP_ENB_K9,
             KYD_OFF := NOT "KYD".TCH_LFT_UP  OR NOT "PDI".MP_ENB_K9,
             AUTO := "APC".AUTOMATIC,
             DC_ON := "SysLog0",
             CON1 := "PDI".EMO AND "PDI".EMS,
             CON2 := NOT "FLT".TCH_LFT_ERR, //TCH_LFT_FU_RDY AND NOT FLT.TCH_LFT_ERR,
             CON3 := NOT "LT".TCH_LFT_DN, 
             CON4 := "PDI".LS_GCH_SW_OUT,   
             CON5 := NOT "PDI".LS_TCH_UP,   
             CON6 := "PDI".LS_TCH_SW_IN OR "PDI".LS_TCH_SW_CLN,                     
             CON7 := "LT".TCH_SW_LOCKED AND "PDI".LS_GCH_UP,    
             CON8 := "PDI".SLS_TCH_LFT AND "PDI".LS_TCH_TILT_0,   
             ITL_OUT := "STA_ITL_CAUSE",
             LT_OUT := "LT".TCH_LFT_UP); 


       "LT".TCH_LFT_UP_REL :=        "PDI".EMO AND "PDI".EMS 
                           AND NOT "FLT".TCH_LFT_ERR 
                         //  AND     TCH_LFT_FU_RDY
                           AND     "PDI".LS_GCH_SW_OUT 
                           AND NOT "PDI".LS_TCH_UP  
                           AND     ("PDI".LS_TCH_SW_IN OR "PDI".LS_TCH_SW_CLN)
                           AND     "LT".TCH_SW_LOCKED
                           AND     "PDI".LS_TCH_TILT_0; 

       // top chamber lift down    
       "CM_ITL_IO"(ADR := 46,                                
             KYD_ON := "KYD".TCH_LFT_DN AND "PDI".MP_ENB_K9,
             KYD_OFF := NOT "KYD".TCH_LFT_DN OR NOT "PDI".MP_ENB_K9,
             AUTO := "APC".AUTOMATIC,
             DC_ON := "SysLog0",
             CON1 := "PDI".EMO AND "PDI".EMS,
             CON2 := NOT "FLT".TCH_LFT_ERR,     // TCH_LFT_FU_RDY AND NOT FLT.TCH_LFT_ERR,
             CON3 := NOT "LT".TCH_LFT_UP,  
             CON4 := "PDI".LS_TEC_FLG_DN,   
             CON5 := NOT "PDI".LS_TCH_DN,   
             CON6 := "PDI".LS_TCH_SW_IN OR "PDI".LS_TCH_SW_CLN,                     
             CON7 := "LT".TCH_SW_LOCKED,    
             CON8 := "PDI".SLS_TCH_LFT AND "PDI".LS_TCH_TILT_0,   
             ITL_OUT:= "STA_ITL_CAUSE",
             LT_OUT := "LT".TCH_LFT_DN); 

